REGION Network 19: DN TRR
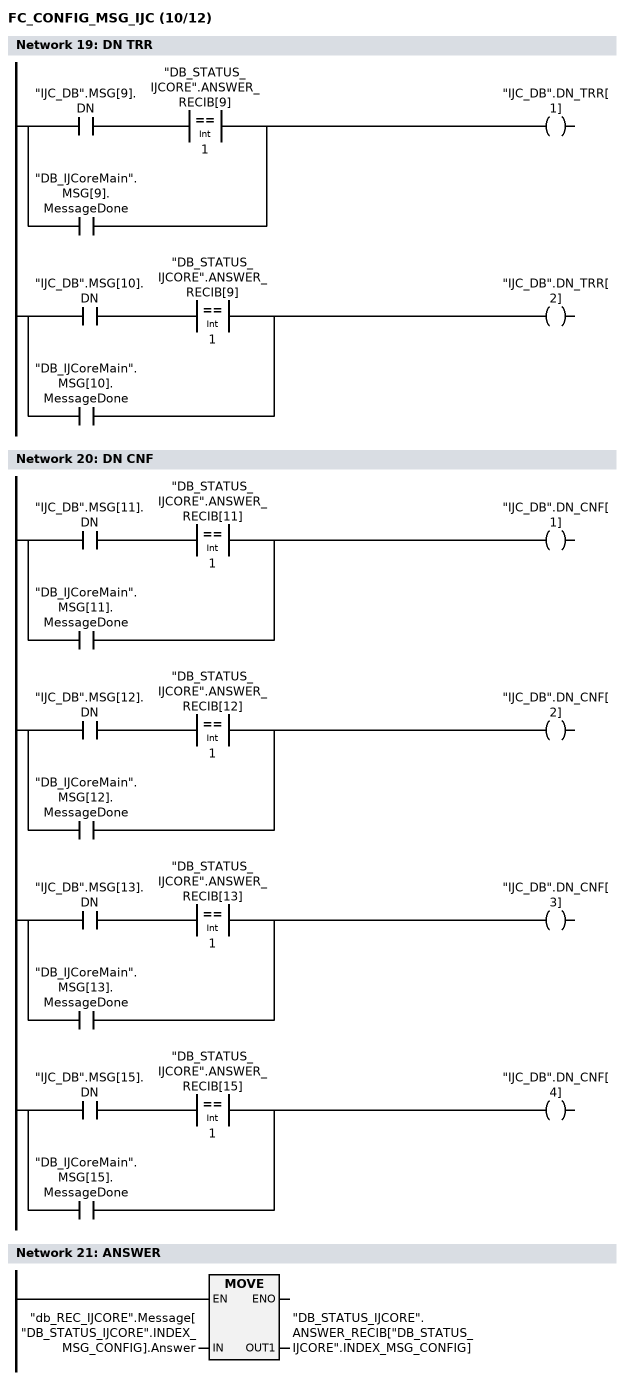
   RUNG wire#powerrail
      Contact( "IJC_DB".MSG[9].DN )
      { S7_Templates := "SrcType := Int" } EQ_Contact(in1 := "DB_STATUS_IJCORE".ANSWER_RECIB[9], in2 := 1)
      wire#w1
      Coil( "IJC_DB".DN_TRR[1] )
   END_RUNG
   RUNG wire#powerrail
      Contact( "DB_IJCoreMain".MSG[9].MessageDone )
   END_RUNG wire#w1
   RUNG wire#powerrail
      Contact( "IJC_DB".MSG[10].DN )
      { S7_Templates := "SrcType := Int" } EQ_Contact(in1 := "DB_STATUS_IJCORE".ANSWER_RECIB[9], in2 := 1)
      wire#w2
      Coil( "IJC_DB".DN_TRR[2] )
   END_RUNG
   RUNG wire#powerrail
      Contact( "DB_IJCoreMain".MSG[10].MessageDone )
   END_RUNG wire#w2
   // the same network as SCL:
   "IJC_DB".DN_TRR[1] := ("IJC_DB".MSG[9].DN AND ("DB_STATUS_IJCORE".ANSWER_RECIB[9] = 1)) OR "DB_IJCoreMain".MSG[9].MessageDone;
   "IJC_DB".DN_TRR[2] := ("IJC_DB".MSG[10].DN AND ("DB_STATUS_IJCORE".ANSWER_RECIB[9] = 1)) OR "DB_IJCoreMain".MSG[10].MessageDone;
END_REGION

REGION Network 20: DN CNF
   RUNG wire#powerrail
      Contact( "IJC_DB".MSG[11].DN )
      { S7_Templates := "SrcType := Int" } EQ_Contact(in1 := "DB_STATUS_IJCORE".ANSWER_RECIB[11], in2 := 1)
      wire#w1
      Coil( "IJC_DB".DN_CNF[1] )
   END_RUNG
   RUNG wire#powerrail
      Contact( "DB_IJCoreMain".MSG[11].MessageDone )
   END_RUNG wire#w1
   RUNG wire#powerrail
      Contact( "IJC_DB".MSG[12].DN )
      { S7_Templates := "SrcType := Int" } EQ_Contact(in1 := "DB_STATUS_IJCORE".ANSWER_RECIB[12], in2 := 1)
      wire#w2
      Coil( "IJC_DB".DN_CNF[2] )
   END_RUNG
   RUNG wire#powerrail
      Contact( "DB_IJCoreMain".MSG[12].MessageDone )
   END_RUNG wire#w2
   RUNG wire#powerrail
      Contact( "IJC_DB".MSG[13].DN )
      { S7_Templates := "SrcType := Int" } EQ_Contact(in1 := "DB_STATUS_IJCORE".ANSWER_RECIB[13], in2 := 1)
      wire#w3
      Coil( "IJC_DB".DN_CNF[3] )
   END_RUNG
   RUNG wire#powerrail
      Contact( "DB_IJCoreMain".MSG[13].MessageDone )
   END_RUNG wire#w3
   RUNG wire#powerrail
      Contact( "IJC_DB".MSG[15].DN )
      { S7_Templates := "SrcType := Int" } EQ_Contact(in1 := "DB_STATUS_IJCORE".ANSWER_RECIB[15], in2 := 1)
      wire#w4
      Coil( "IJC_DB".DN_CNF[4] )
   END_RUNG
   RUNG wire#powerrail
      Contact( "DB_IJCoreMain".MSG[15].MessageDone )
   END_RUNG wire#w4
   // the same network as SCL:
   "IJC_DB".DN_CNF[1] := ("IJC_DB".MSG[11].DN AND ("DB_STATUS_IJCORE".ANSWER_RECIB[11] = 1)) OR "DB_IJCoreMain".MSG[11].MessageDone;
   "IJC_DB".DN_CNF[2] := ("IJC_DB".MSG[12].DN AND ("DB_STATUS_IJCORE".ANSWER_RECIB[12] = 1)) OR "DB_IJCoreMain".MSG[12].MessageDone;
   "IJC_DB".DN_CNF[3] := ("IJC_DB".MSG[13].DN AND ("DB_STATUS_IJCORE".ANSWER_RECIB[13] = 1)) OR "DB_IJCoreMain".MSG[13].MessageDone;
   "IJC_DB".DN_CNF[4] := ("IJC_DB".MSG[15].DN AND ("DB_STATUS_IJCORE".ANSWER_RECIB[15] = 1)) OR "DB_IJCoreMain".MSG[15].MessageDone;
END_REGION

REGION Network 21: ANSWER
   RUNG wire#powerrail
      Move(in := "db_REC_IJCORE".Message["DB_STATUS_IJCORE".INDEX_MSG_CONFIG].Answer, out1 => "DB_STATUS_IJCORE".ANSWER_RECIB["DB_STATUS_IJCORE".INDEX_MSG_CONFIG])
   END_RUNG
   // the same network as SCL:
   "DB_STATUS_IJCORE".ANSWER_RECIB["DB_STATUS_IJCORE".INDEX_MSG_CONFIG] := "db_REC_IJCORE".Message["DB_STATUS_IJCORE".INDEX_MSG_CONFIG].Answer;
END_REGION

REGION Network 22: ANSWER NFP
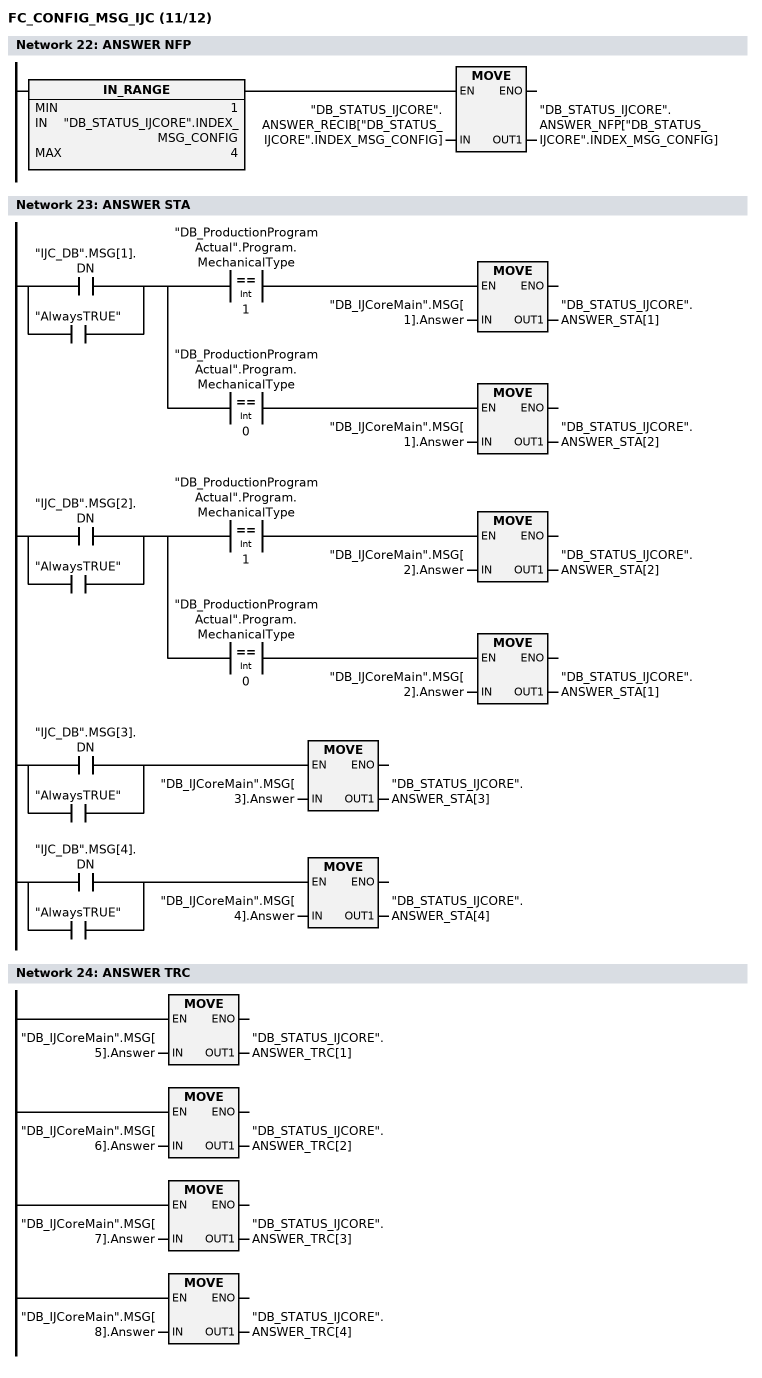
   RUNG wire#powerrail
      { S7_Templates := "SrcType := DInt" } InRange(min := 1, in := "DB_STATUS_IJCORE".INDEX_MSG_CONFIG, max := 4)
      Move(in := "DB_STATUS_IJCORE".ANSWER_RECIB["DB_STATUS_IJCORE".INDEX_MSG_CONFIG], out1 => "DB_STATUS_IJCORE".ANSWER_NFP["DB_STATUS_IJCORE".INDEX_MSG_CONFIG])
   END_RUNG
   // the same network as SCL:
   IF (1 <= "DB_STATUS_IJCORE".INDEX_MSG_CONFIG) AND ("DB_STATUS_IJCORE".INDEX_MSG_CONFIG <= 4) THEN
       "DB_STATUS_IJCORE".ANSWER_NFP["DB_STATUS_IJCORE".INDEX_MSG_CONFIG] := "DB_STATUS_IJCORE".ANSWER_RECIB["DB_STATUS_IJCORE".INDEX_MSG_CONFIG];
   END_IF;
END_REGION

REGION Network 23: ANSWER STA
   RUNG wire#powerrail
      Contact( "IJC_DB".MSG[1].DN )
      wire#w1
      { S7_Templates := "SrcType := Int" } EQ_Contact(in1 := "DB_ProductionProgramActual".Program.MechanicalType, in2 := 1)
      Move(in := "DB_IJCoreMain".MSG[1].Answer, out1 => "DB_STATUS_IJCORE".ANSWER_STA[1])
   END_RUNG
   RUNG wire#powerrail
      Contact( "AlwaysTRUE" )
   END_RUNG wire#w1
   RUNG wire#w1
      { S7_Templates := "SrcType := Int" } EQ_Contact(in1 := "DB_ProductionProgramActual".Program.MechanicalType, in2 := 0)
      Move(in := "DB_IJCoreMain".MSG[1].Answer, out1 => "DB_STATUS_IJCORE".ANSWER_STA[2])
   END_RUNG
   RUNG wire#powerrail
      Contact( "IJC_DB".MSG[2].DN )
      wire#w2
      { S7_Templates := "SrcType := Int" } EQ_Contact(in1 := "DB_ProductionProgramActual".Program.MechanicalType, in2 := 1)
      Move(in := "DB_IJCoreMain".MSG[2].Answer, out1 => "DB_STATUS_IJCORE".ANSWER_STA[2])
   END_RUNG
   RUNG wire#powerrail
      Contact( "AlwaysTRUE" )
   END_RUNG wire#w2
   RUNG wire#w2
      { S7_Templates := "SrcType := Int" } EQ_Contact(in1 := "DB_ProductionProgramActual".Program.MechanicalType, in2 := 0)
      Move(in := "DB_IJCoreMain".MSG[2].Answer, out1 => "DB_STATUS_IJCORE".ANSWER_STA[1])
   END_RUNG
   RUNG wire#powerrail
      Contact( "IJC_DB".MSG[3].DN )
      wire#w3
      Move(in := "DB_IJCoreMain".MSG[3].Answer, out1 => "DB_STATUS_IJCORE".ANSWER_STA[3])
   END_RUNG
   RUNG wire#powerrail
      Contact( "AlwaysTRUE" )
   END_RUNG wire#w3
   RUNG wire#powerrail
      Contact( "IJC_DB".MSG[4].DN )
      wire#w4
      Move(in := "DB_IJCoreMain".MSG[4].Answer, out1 => "DB_STATUS_IJCORE".ANSWER_STA[4])
   END_RUNG
   RUNG wire#powerrail
      Contact( "AlwaysTRUE" )
   END_RUNG wire#w4
   // the same network as SCL:
   #_w1 := "IJC_DB".MSG[1].DN OR "AlwaysTRUE";
   IF #_w1 AND ("DB_ProductionProgramActual".Program.MechanicalType = 1) THEN
       "DB_STATUS_IJCORE".ANSWER_STA[1] := "DB_IJCoreMain".MSG[1].Answer;
   END_IF;
   IF #_w1 AND ("DB_ProductionProgramActual".Program.MechanicalType = 0) THEN
       "DB_STATUS_IJCORE".ANSWER_STA[2] := "DB_IJCoreMain".MSG[1].Answer;
   END_IF;
   #_w2 := "IJC_DB".MSG[2].DN OR "AlwaysTRUE";
   IF #_w2 AND ("DB_ProductionProgramActual".Program.MechanicalType = 1) THEN
       "DB_STATUS_IJCORE".ANSWER_STA[2] := "DB_IJCoreMain".MSG[2].Answer;
   END_IF;
   IF #_w2 AND ("DB_ProductionProgramActual".Program.MechanicalType = 0) THEN
       "DB_STATUS_IJCORE".ANSWER_STA[1] := "DB_IJCoreMain".MSG[2].Answer;
   END_IF;
   IF "IJC_DB".MSG[3].DN OR "AlwaysTRUE" THEN
       "DB_STATUS_IJCORE".ANSWER_STA[3] := "DB_IJCoreMain".MSG[3].Answer;
   END_IF;
   IF "IJC_DB".MSG[4].DN OR "AlwaysTRUE" THEN
       "DB_STATUS_IJCORE".ANSWER_STA[4] := "DB_IJCoreMain".MSG[4].Answer;
   END_IF;
END_REGION

REGION Network 24: ANSWER TRC
   RUNG wire#powerrail
      Move(in := "DB_IJCoreMain".MSG[5].Answer, out1 => "DB_STATUS_IJCORE".ANSWER_TRC[1])
   END_RUNG
   RUNG wire#powerrail
      Move(in := "DB_IJCoreMain".MSG[6].Answer, out1 => "DB_STATUS_IJCORE".ANSWER_TRC[2])
   END_RUNG
   RUNG wire#powerrail
      Move(in := "DB_IJCoreMain".MSG[7].Answer, out1 => "DB_STATUS_IJCORE".ANSWER_TRC[3])
   END_RUNG
   RUNG wire#powerrail
      Move(in := "DB_IJCoreMain".MSG[8].Answer, out1 => "DB_STATUS_IJCORE".ANSWER_TRC[4])
   END_RUNG
   // the same network as SCL:
   "DB_STATUS_IJCORE".ANSWER_TRC[1] := "DB_IJCoreMain".MSG[5].Answer;
   "DB_STATUS_IJCORE".ANSWER_TRC[2] := "DB_IJCoreMain".MSG[6].Answer;
   "DB_STATUS_IJCORE".ANSWER_TRC[3] := "DB_IJCoreMain".MSG[7].Answer;
   "DB_STATUS_IJCORE".ANSWER_TRC[4] := "DB_IJCoreMain".MSG[8].Answer;
END_REGION

REGION Network 25: STATUS MSG TRC
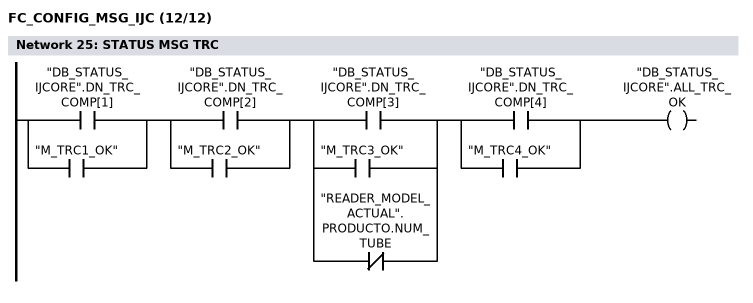
   RUNG wire#powerrail
      Contact( "DB_STATUS_IJCORE".DN_TRC_COMP[1] )
      wire#w1
      Contact( "DB_STATUS_IJCORE".DN_TRC_COMP[2] )
      wire#w2
      Contact( "DB_STATUS_IJCORE".DN_TRC_COMP[3] )
      wire#w3
      Contact( "DB_STATUS_IJCORE".DN_TRC_COMP[4] )
      wire#w4
      Coil( "DB_STATUS_IJCORE".ALL_TRC_OK )
   END_RUNG
   RUNG wire#powerrail
      Contact( "M_TRC1_OK" )
   END_RUNG wire#w1
   RUNG wire#w1
      Contact( "M_TRC2_OK" )
   END_RUNG wire#w2
   RUNG wire#w2
      Contact( "M_TRC3_OK" )
   END_RUNG wire#w3
   RUNG wire#w2
      I_Contact( "READER_MODEL_ACTUAL".PRODUCTO.NUM_TUBE )
   END_RUNG wire#w3
   RUNG wire#w3
      Contact( "M_TRC4_OK" )
   END_RUNG wire#w4
   // the same network as SCL:
   "DB_STATUS_IJCORE".ALL_TRC_OK := ("DB_STATUS_IJCORE".DN_TRC_COMP[1] OR "M_TRC1_OK") AND ("DB_STATUS_IJCORE".DN_TRC_COMP[2] OR "M_TRC2_OK") AND ("DB_STATUS_IJCORE".DN_TRC_COMP[3] OR "M_TRC3_OK" OR NOT "READER_MODEL_ACTUAL".PRODUCTO.NUM_TUBE) AND ("DB_STATUS_IJCORE".DN_TRC_COMP[4] OR "M_TRC4_OK");
END_REGION
END_FUNCTION

FUNCTION_BLOCK "AWAKE_SIGNAL"   // FB1002, LAD
TITLE = Awake signal
{ S7_Optimized_Access := 'TRUE' }
VERSION : 0.1
// This function supervise Awake signal, 
// - Awake signal is to test communication between PLC and IJCORE. 
// - Awake signal is set to 1 by PLC and set to -1 by IJCORE alternatively.
// - first PLC check if awake signal is different of 1, if it is, PLC launch timer T1 
//  (1s<T1<10s). at the end of this temporisation, PLC set awake signal to 1 and 
//  launch Timer 2. 
// - if IJCORE don't set awake signal to -1 before the end of timer 2,PLC generate  
//   Time out fault for awake signal.
// stored: AutoNumber false, IsIECCheckEnabled false, IsRetainMemResEnabled false, MemoryReserve 100, SetENOAutomatically false, UDAEnableTagReadback false
   VAR_INPUT
      ack_error : Bool;   // Acknowledge button
   END_VAR
   VAR_OUTPUT
      State_com : SInt;   // State of communication : 0 no communication 1: communication lost 2 : good communication
   END_VAR
   VAR RETAIN
      T1PresetValue : Time := T#1S;   // Bit of life Timer 1 preset value
      T2PresetValue : Time := T#60S;   // Bit of Life Timer 2 preset value
   END_VAR
   VAR
      AwSignalTimeOutFault : Bool := 0;   // Awake signal time out fault
      Reset_Counters : Bool;   // Signal to reset counter
      Restart_Counter_bit_of_life : USInt := 0;   // Number of restart bit of life
      NB_Bit_of_Life : Bool;   // Number bit of life
      number_restart : DInt;   // Number restart communication
      check_restart : Bool;   // Memo to check restart communication
      t13 : TON_TIME;
      t16 { S7_SetPoint := 'True'} : TON_TIME;
      t5 { S7_SetPoint := 'True'} : TON_TIME;
      t4 { S7_SetPoint := 'True'} : TON_TIME;
   END_VAR
   VAR CONSTANT
      Trestart : Time := T#200ms;   // Timer when IJCore replies normally
      T3 : Time := T#2s;   // Timer when IJCore blocks a short period of time
   END_VAR
   VAR_TEMP   // added for the SCL form of the ladder/FBD networks
      _w1 : Bool;
   END_VAR
BEGIN

REGION Network 1: - if awake signal is -1 then launch timer 1
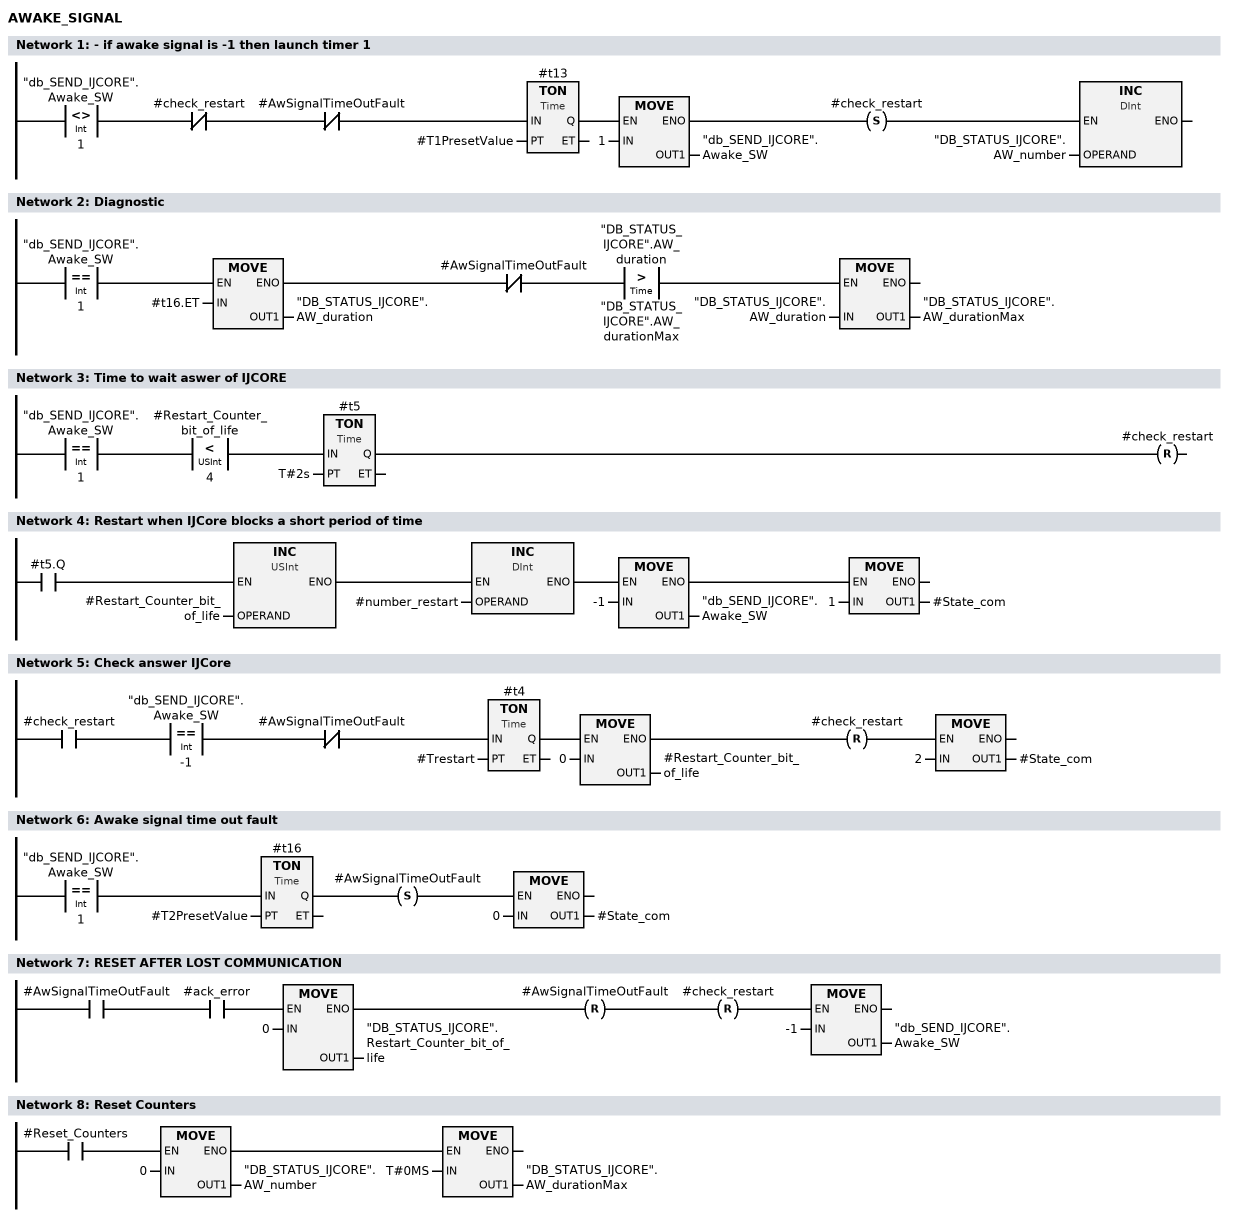
   RUNG wire#powerrail
      { S7_Templates := "SrcType := Int" } NE_Contact(in1 := "db_SEND_IJCORE".Awake_SW, in2 := 1)
      I_Contact( #check_restart )
      I_Contact( #AwSignalTimeOutFault )
      { S7_Templates := "time_type := Time" } #t13.TON(pt := #T1PresetValue, et =>)
      Move(in := 1, out1 => "db_SEND_IJCORE".Awake_SW)
      S_Coil( #check_restart )
      { S7_Templates := "DestType := DInt" } Inc( "DB_STATUS_IJCORE".AW_number )
   END_RUNG
   // the same network as SCL:
   #t13(IN := ("db_SEND_IJCORE".Awake_SW <> 1) AND NOT #check_restart AND NOT #AwSignalTimeOutFault,   // TON
        PT := #T1PresetValue);
   IF #t13.Q THEN
       "db_SEND_IJCORE".Awake_SW := 1;
       #check_restart := TRUE;
       "DB_STATUS_IJCORE".AW_number := "DB_STATUS_IJCORE".AW_number + 1;
   END_IF;
END_REGION

REGION Network 2: Diagnostic
   RUNG wire#powerrail
      { S7_Templates := "SrcType := Int" } EQ_Contact(in1 := "db_SEND_IJCORE".Awake_SW, in2 := 1)
      Move(in := #t16.ET, out1 => "DB_STATUS_IJCORE".AW_duration)
      I_Contact( #AwSignalTimeOutFault )
      { S7_Templates := "SrcType := Time" } GT_Contact(in1 := "DB_STATUS_IJCORE".AW_duration, in2 := "DB_STATUS_IJCORE".AW_durationMax)
      Move(in := "DB_STATUS_IJCORE".AW_duration, out1 => "DB_STATUS_IJCORE".AW_durationMax)
   END_RUNG
   // the same network as SCL:
   #_w1 := "db_SEND_IJCORE".Awake_SW = 1;
   IF #_w1 THEN "DB_STATUS_IJCORE".AW_duration := #t16.ET; END_IF;
   IF #_w1 AND NOT #AwSignalTimeOutFault AND ("DB_STATUS_IJCORE".AW_duration > "DB_STATUS_IJCORE".AW_durationMax) THEN
       "DB_STATUS_IJCORE".AW_durationMax := "DB_STATUS_IJCORE".AW_duration;
   END_IF;
END_REGION

REGION Network 3: Time to wait aswer of IJCORE
   RUNG wire#powerrail
      { S7_Templates := "SrcType := Int" } EQ_Contact(in1 := "db_SEND_IJCORE".Awake_SW, in2 := 1)
      { S7_Templates := "SrcType := USInt" } LT_Contact(in1 := #Restart_Counter_bit_of_life, in2 := 4)
      { S7_Templates := "time_type := Time" } #t5.TON(pt := T#2s, et =>)
      R_Coil( #check_restart )
   END_RUNG
   // the same network as SCL:
   #t5(IN := ("db_SEND_IJCORE".Awake_SW = 1) AND (#Restart_Counter_bit_of_life < 4), PT := T#2s);   // TON
   IF #t5.Q THEN #check_restart := FALSE; END_IF;
END_REGION

REGION Network 4: Restart when IJCore blocks a short period of time
   RUNG wire#powerrail
      Contact( #t5.Q )
      { S7_Templates := "DestType := USInt" } Inc( #Restart_Counter_bit_of_life )
      { S7_Templates := "DestType := DInt" } Inc( #number_restart )
      Move(in := -1, out1 => "db_SEND_IJCORE".Awake_SW)
      Move(in := 1, out1 => #State_com)
   END_RUNG
   // the same network as SCL:
   IF #t5.Q THEN
       #Restart_Counter_bit_of_life := #Restart_Counter_bit_of_life + 1;
       #number_restart := #number_restart + 1;
       "db_SEND_IJCORE".Awake_SW := -1;
       #State_com := 1;
   END_IF;
END_REGION

REGION Network 5: Check answer IJCore
   RUNG wire#powerrail
      Contact( #check_restart )
      { S7_Templates := "SrcType := Int" } EQ_Contact(in1 := "db_SEND_IJCORE".Awake_SW, in2 := -1)
      I_Contact( #AwSignalTimeOutFault )
      { S7_Templates := "time_type := Time" } #t4.TON(pt := #Trestart, et =>)
      Move(in := 0, out1 => #Restart_Counter_bit_of_life)
      R_Coil( #check_restart )
      Move(in := 2, out1 => #State_com)
   END_RUNG
   // the same network as SCL:
   #t4(IN := #check_restart AND ("db_SEND_IJCORE".Awake_SW = (-1)) AND NOT #AwSignalTimeOutFault,   // TON
       PT := #Trestart);
   IF #t4.Q THEN
       #Restart_Counter_bit_of_life := 0;
       #check_restart := FALSE;
       #State_com := 2;
   END_IF;
END_REGION

REGION Network 6: Awake signal time out fault
   RUNG wire#powerrail
      { S7_Templates := "SrcType := Int" } EQ_Contact(in1 := "db_SEND_IJCORE".Awake_SW, in2 := 1)
      { S7_Templates := "time_type := Time" } #t16.TON(pt := #T2PresetValue, et =>)
      S_Coil( #AwSignalTimeOutFault )
      Move(in := 0, out1 => #State_com)
   END_RUNG
   // the same network as SCL:
   #t16(IN := "db_SEND_IJCORE".Awake_SW = 1, PT := #T2PresetValue);   // TON
   IF #t16.Q THEN
       #AwSignalTimeOutFault := TRUE;
       #State_com := 0;
   END_IF;
END_REGION

REGION Network 7: RESET AFTER LOST COMMUNICATION
   RUNG wire#powerrail
      Contact( #AwSignalTimeOutFault )
      Contact( #ack_error )
      Move(in := 0, out1 => "DB_STATUS_IJCORE".Restart_Counter_bit_of_life)
      R_Coil( #AwSignalTimeOutFault )
      R_Coil( #check_restart )
      Move(in := -1, out1 => "db_SEND_IJCORE".Awake_SW)
   END_RUNG
   // the same network as SCL:
   IF #AwSignalTimeOutFault AND #ack_error THEN "DB_STATUS_IJCORE".Restart_Counter_bit_of_life := 0; END_IF;
   #_w1 := #AwSignalTimeOutFault AND #ack_error;
   IF #_w1 THEN
       #AwSignalTimeOutFault := FALSE;
       #check_restart := FALSE;
       "db_SEND_IJCORE".Awake_SW := -1;
   END_IF;
END_REGION

REGION Network 8: Reset Counters
   RUNG wire#powerrail
      Contact( #Reset_Counters )
      Move(in := 0, out1 => "DB_STATUS_IJCORE".AW_number)
      Move(in := T#0MS, out1 => "DB_STATUS_IJCORE".AW_durationMax)
   END_RUNG
   // the same network as SCL:
   IF #Reset_Counters THEN
       "DB_STATUS_IJCORE".AW_number := 0;
       "DB_STATUS_IJCORE".AW_durationMax := T#0MS;
   END_IF;
END_REGION
END_FUNCTION_BLOCK

FUNCTION_BLOCK "IJCoreMain"   // FB1000, LAD
TITLE = IJCore Main
{ S7_Optimized_Access := 'TRUE' }
VERSION : 0.1
// stored: AutoNumber false, IsIECCheckEnabled false, IsRetainMemResEnabled false, MemoryReserve 100, SetENOAutomatically false, UDAEnableTagReadback false
   VAR
      Enable : Bool;
      Mode : UInt;
      Indicator : Int;
      AlarmReset : Bool;
      AWAKE_SIGNAL { S7_SetPoint := 'True'} : "AWAKE_SIGNAL";
      MSG : Array[1..20] of "IJCoreMessageProcotol";
      NFP { S7_SetPoint := 'True'} : Array[1..4] of String[30];
   END_VAR
   VAR_TEMP
      MessageDone : Bool;
      Answer : DInt;
      Fault : DInt;
   END_VAR
   VAR CONSTANT
      STA : Int := 5;
      CNF : Int := 1;
      TRC : Int := 13;
      PFC : Int := 9;
      TRR : Int := 7;
   END_VAR
BEGIN

REGION Network 1
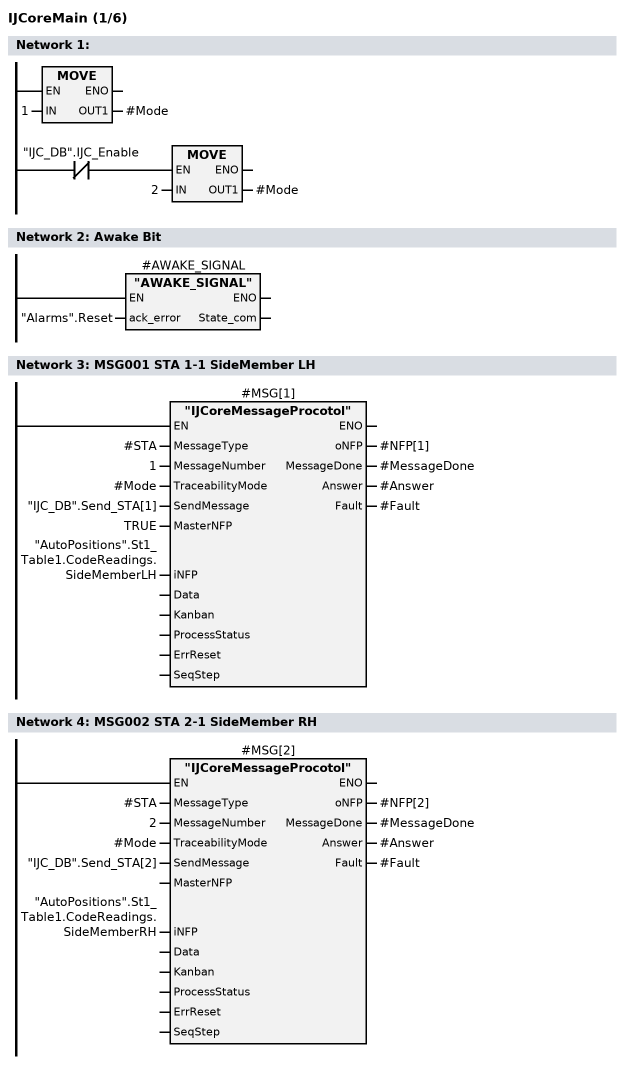
   RUNG wire#powerrail
      Move(in := 1, out1 => #Mode)
   END_RUNG
   RUNG wire#powerrail
      I_Contact( "IJC_DB".IJC_Enable )
      Move(in := 2, out1 => #Mode)
   END_RUNG
   // the same network as SCL:
   #Mode := 1;
   IF NOT "IJC_DB".IJC_Enable THEN #Mode := 2; END_IF;
END_REGION

REGION Network 2: Awake Bit
   RUNG wire#powerrail
      #AWAKE_SIGNAL(ack_error := "Alarms".Reset, State_com =>)
   END_RUNG
   // the same network as SCL:
   #AWAKE_SIGNAL(ack_error := "Alarms".Reset);   // "AWAKE_SIGNAL"
END_REGION

REGION Network 3: MSG001 STA 1-1 SideMember LH
   RUNG wire#powerrail
      #MSG[1](MessageType := #STA, MessageNumber := 1, TraceabilityMode := #Mode, SendMessage := "IJC_DB".Send_STA[1], MasterNFP := TRUE, iNFP := "AutoPositions".St1_Table1.CodeReadings.SideMemberLH, Data :=, Kanban :=, ProcessStatus :=, ErrReset :=, SeqStep :=, oNFP => #NFP[1], MessageDone => #MessageDone, Answer => #Answer, Fault => #Fault)
   END_RUNG
   // the same network as SCL:
   #MSG[1](MessageType := #STA,   // "IJCoreMessageProcotol"
           MessageNumber := 1,
           TraceabilityMode := #Mode,
           SendMessage := "IJC_DB".Send_STA[1],
           MasterNFP := TRUE,
           iNFP := "AutoPositions".St1_Table1.CodeReadings.SideMemberLH,
           oNFP => #NFP[1],
           MessageDone => #MessageDone,
           Answer => #Answer,
           Fault => #Fault);
END_REGION

REGION Network 4: MSG002 STA 2-1 SideMember RH
   RUNG wire#powerrail
      #MSG[2](MessageType := #STA, MessageNumber := 2, TraceabilityMode := #Mode, SendMessage := "IJC_DB".Send_STA[2], MasterNFP :=, iNFP := "AutoPositions".St1_Table1.CodeReadings.SideMemberRH, Data :=, Kanban :=, ProcessStatus :=, ErrReset :=, SeqStep :=, oNFP => #NFP[2], MessageDone => #MessageDone, Answer => #Answer, Fault => #Fault)
   END_RUNG
   // the same network as SCL:
   #MSG[2](MessageType := #STA,   // "IJCoreMessageProcotol"
           MessageNumber := 2,
           TraceabilityMode := #Mode,
           SendMessage := "IJC_DB".Send_STA[2],
           iNFP := "AutoPositions".St1_Table1.CodeReadings.SideMemberRH,
           oNFP => #NFP[2],
           MessageDone => #MessageDone,
           Answer => #Answer,
           Fault => #Fault);
END_REGION

REGION Network 5: MSG003 STA 3-1 Front Tube
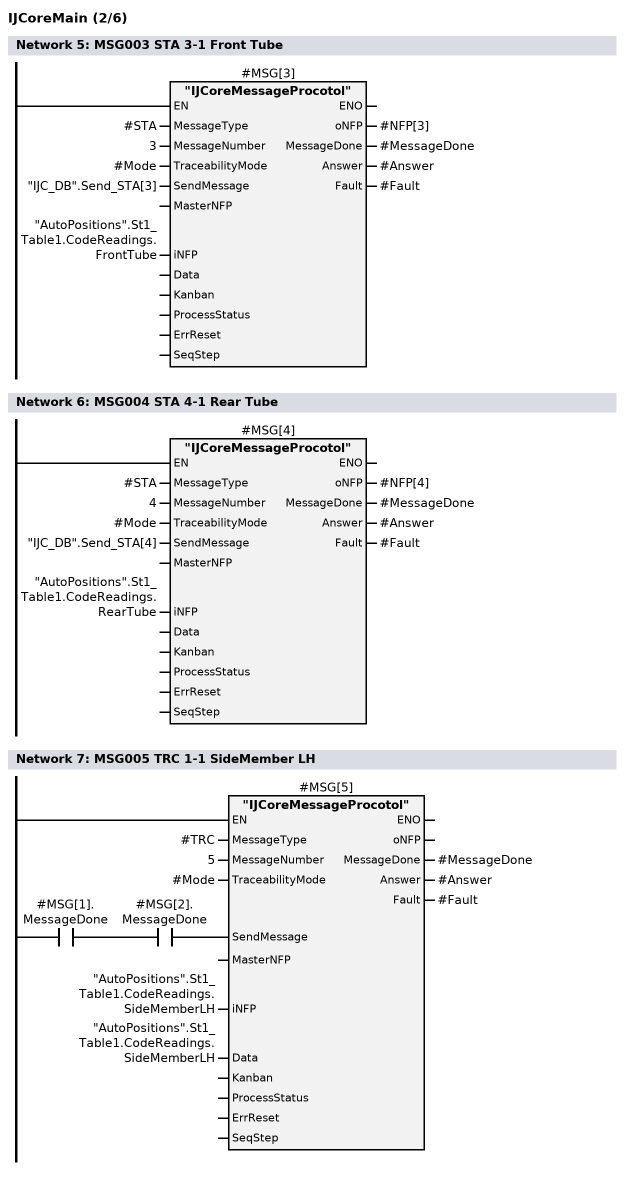
   RUNG wire#powerrail
      #MSG[3](MessageType := #STA, MessageNumber := 3, TraceabilityMode := #Mode, SendMessage := "IJC_DB".Send_STA[3], MasterNFP :=, iNFP := "AutoPositions".St1_Table1.CodeReadings.FrontTube, Data :=, Kanban :=, ProcessStatus :=, ErrReset :=, SeqStep :=, oNFP => #NFP[3], MessageDone => #MessageDone, Answer => #Answer, Fault => #Fault)
   END_RUNG
   // the same network as SCL:
   #MSG[3](MessageType := #STA,   // "IJCoreMessageProcotol"
           MessageNumber := 3,
           TraceabilityMode := #Mode,
           SendMessage := "IJC_DB".Send_STA[3],
           iNFP := "AutoPositions".St1_Table1.CodeReadings.FrontTube,
           oNFP => #NFP[3],
           MessageDone => #MessageDone,
           Answer => #Answer,
           Fault => #Fault);
END_REGION

REGION Network 6: MSG004 STA 4-1 Rear Tube
   RUNG wire#powerrail
      #MSG[4](MessageType := #STA, MessageNumber := 4, TraceabilityMode := #Mode, SendMessage := "IJC_DB".Send_STA[4], MasterNFP :=, iNFP := "AutoPositions".St1_Table1.CodeReadings.RearTube, Data :=, Kanban :=, ProcessStatus :=, ErrReset :=, SeqStep :=, oNFP => #NFP[4], MessageDone => #MessageDone, Answer => #Answer, Fault => #Fault)
   END_RUNG
   // the same network as SCL:
   #MSG[4](MessageType := #STA,   // "IJCoreMessageProcotol"
           MessageNumber := 4,
           TraceabilityMode := #Mode,
           SendMessage := "IJC_DB".Send_STA[4],
           iNFP := "AutoPositions".St1_Table1.CodeReadings.RearTube,
           oNFP => #NFP[4],
           MessageDone => #MessageDone,
           Answer => #Answer,
           Fault => #Fault);
END_REGION

REGION Network 7: MSG005 TRC 1-1 SideMember LH
   RUNG wire#powerrail
      #MSG[5](SendMessage := wire#w1, MessageType := #TRC, MessageNumber := 5, TraceabilityMode := #Mode, MasterNFP :=, iNFP := "AutoPositions".St1_Table1.CodeReadings.SideMemberLH, Data := "AutoPositions".St1_Table1.CodeReadings.SideMemberLH, Kanban :=, ProcessStatus :=, ErrReset :=, SeqStep :=, oNFP =>, MessageDone => #MessageDone, Answer => #Answer, Fault => #Fault)
   END_RUNG
   RUNG wire#powerrail
      Contact( #MSG[1].MessageDone )
      Contact( #MSG[2].MessageDone )
   END_RUNG wire#w1
   // the same network as SCL:
   #MSG[5](MessageType := #TRC,   // "IJCoreMessageProcotol"
           MessageNumber := 5,
           TraceabilityMode := #Mode,
           SendMessage := #MSG[1].MessageDone AND #MSG[2].MessageDone,
           iNFP := "AutoPositions".St1_Table1.CodeReadings.SideMemberLH,
           Data := "AutoPositions".St1_Table1.CodeReadings.SideMemberLH,
           MessageDone => #MessageDone,
           Answer => #Answer,
           Fault => #Fault);
END_REGION

REGION Network 8: MSG006 TRC 1-2 SideMember RH
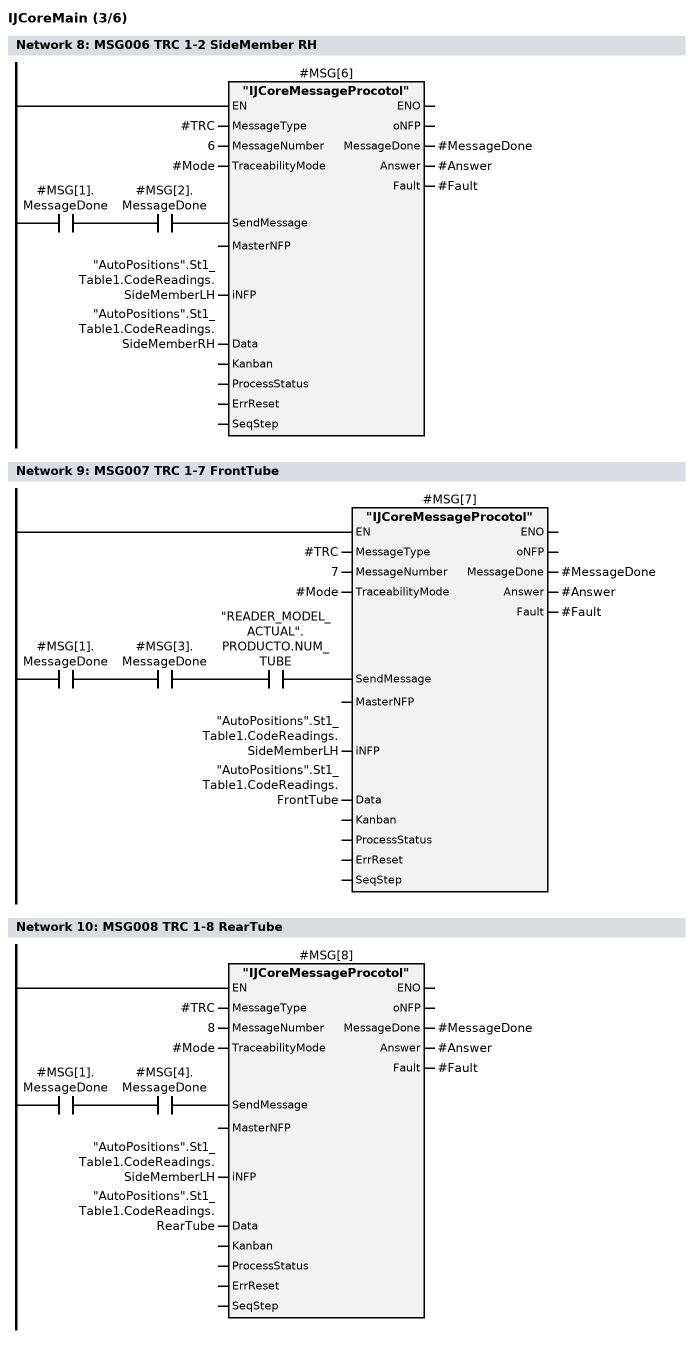
   RUNG wire#powerrail
      #MSG[6](SendMessage := wire#w1, MessageType := #TRC, MessageNumber := 6, TraceabilityMode := #Mode, MasterNFP :=, iNFP := "AutoPositions".St1_Table1.CodeReadings.SideMemberLH, Data := "AutoPositions".St1_Table1.CodeReadings.SideMemberRH, Kanban :=, ProcessStatus :=, ErrReset :=, SeqStep :=, oNFP =>, MessageDone => #MessageDone, Answer => #Answer, Fault => #Fault)
   END_RUNG
   RUNG wire#powerrail
      Contact( #MSG[1].MessageDone )
      Contact( #MSG[2].MessageDone )
   END_RUNG wire#w1
   // the same network as SCL:
   #MSG[6](MessageType := #TRC,   // "IJCoreMessageProcotol"
           MessageNumber := 6,
           TraceabilityMode := #Mode,
           SendMessage := #MSG[1].MessageDone AND #MSG[2].MessageDone,
           iNFP := "AutoPositions".St1_Table1.CodeReadings.SideMemberLH,
           Data := "AutoPositions".St1_Table1.CodeReadings.SideMemberRH,
           MessageDone => #MessageDone,
           Answer => #Answer,
           Fault => #Fault);
END_REGION

REGION Network 9: MSG007 TRC 1-7 FrontTube
   RUNG wire#powerrail
      #MSG[7](SendMessage := wire#w1, MessageType := #TRC, MessageNumber := 7, TraceabilityMode := #Mode, MasterNFP :=, iNFP := "AutoPositions".St1_Table1.CodeReadings.SideMemberLH, Data := "AutoPositions".St1_Table1.CodeReadings.FrontTube, Kanban :=, ProcessStatus :=, ErrReset :=, SeqStep :=, oNFP =>, MessageDone => #MessageDone, Answer => #Answer, Fault => #Fault)
   END_RUNG
   RUNG wire#powerrail
      Contact( #MSG[1].MessageDone )
      Contact( #MSG[3].MessageDone )
      Contact( "READER_MODEL_ACTUAL".PRODUCTO.NUM_TUBE )
   END_RUNG wire#w1
   // the same network as SCL:
   #MSG[7](MessageType := #TRC,   // "IJCoreMessageProcotol"
           MessageNumber := 7,
           TraceabilityMode := #Mode,
           SendMessage := #MSG[1].MessageDone AND #MSG[3].MessageDone AND "READER_MODEL_ACTUAL".PRODUCTO.NUM_TUBE,
           iNFP := "AutoPositions".St1_Table1.CodeReadings.SideMemberLH,
           Data := "AutoPositions".St1_Table1.CodeReadings.FrontTube,
           MessageDone => #MessageDone,
           Answer => #Answer,
           Fault => #Fault);
END_REGION

REGION Network 10: MSG008 TRC 1-8 RearTube
   RUNG wire#powerrail
      #MSG[8](SendMessage := wire#w1, MessageType := #TRC, MessageNumber := 8, TraceabilityMode := #Mode, MasterNFP :=, iNFP := "AutoPositions".St1_Table1.CodeReadings.SideMemberLH, Data := "AutoPositions".St1_Table1.CodeReadings.RearTube, Kanban :=, ProcessStatus :=, ErrReset :=, SeqStep :=, oNFP =>, MessageDone => #MessageDone, Answer => #Answer, Fault => #Fault)
   END_RUNG
   RUNG wire#powerrail
      Contact( #MSG[1].MessageDone )
      Contact( #MSG[4].MessageDone )
   END_RUNG wire#w1
   // the same network as SCL:
   #MSG[8](MessageType := #TRC,   // "IJCoreMessageProcotol"
           MessageNumber := 8,
           TraceabilityMode := #Mode,
           SendMessage := #MSG[1].MessageDone AND #MSG[4].MessageDone,
           iNFP := "AutoPositions".St1_Table1.CodeReadings.SideMemberLH,
           Data := "AutoPositions".St1_Table1.CodeReadings.RearTube,
           MessageDone => #MessageDone,
           Answer => #Answer,
           Fault => #Fault);
END_REGION

REGION Network 11: MSG009 TRR 1-1 Results of riveting
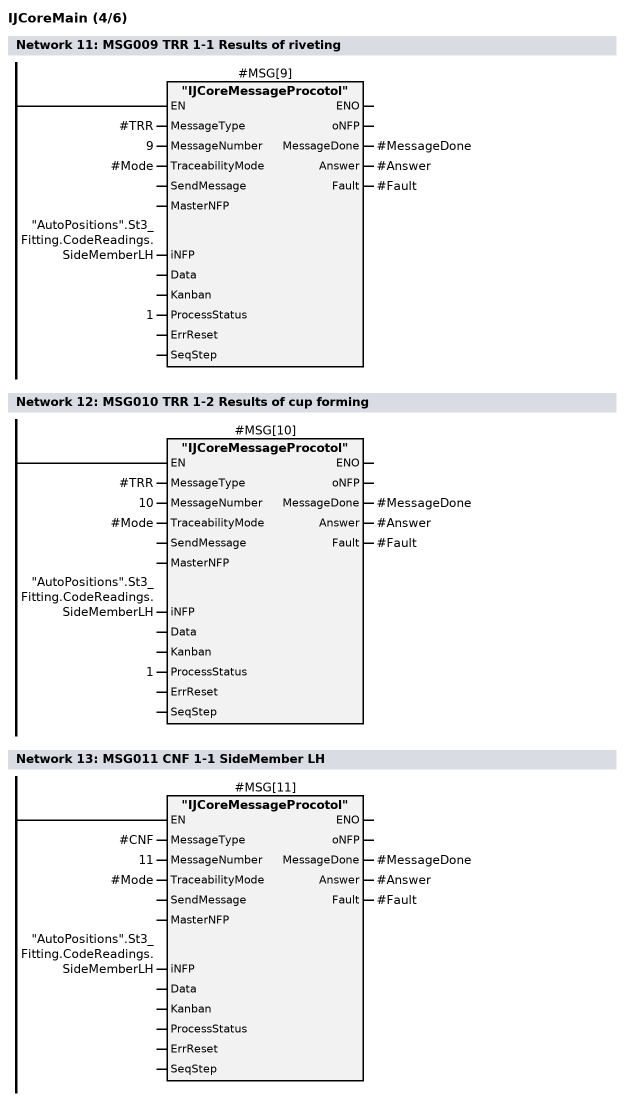
   RUNG wire#powerrail
      #MSG[9](MessageType := #TRR, MessageNumber := 9, TraceabilityMode := #Mode, SendMessage :=, MasterNFP :=, iNFP := "AutoPositions".St3_Fitting.CodeReadings.SideMemberLH, Data :=, Kanban :=, ProcessStatus := 1, ErrReset :=, SeqStep :=, oNFP =>, MessageDone => #MessageDone, Answer => #Answer, Fault => #Fault)
   END_RUNG
   // the same network as SCL:
   #MSG[9](MessageType := #TRR,   // "IJCoreMessageProcotol"
           MessageNumber := 9,
           TraceabilityMode := #Mode,
           iNFP := "AutoPositions".St3_Fitting.CodeReadings.SideMemberLH,
           ProcessStatus := 1,
           MessageDone => #MessageDone,
           Answer => #Answer,
           Fault => #Fault);
END_REGION

REGION Network 12: MSG010 TRR 1-2 Results of cup forming
   RUNG wire#powerrail
      #MSG[10](MessageType := #TRR, MessageNumber := 10, TraceabilityMode := #Mode, SendMessage :=, MasterNFP :=, iNFP := "AutoPositions".St3_Fitting.CodeReadings.SideMemberLH, Data :=, Kanban :=, ProcessStatus := 1, ErrReset :=, SeqStep :=, oNFP =>, MessageDone => #MessageDone, Answer => #Answer, Fault => #Fault)
   END_RUNG
   // the same network as SCL:
   #MSG[10](MessageType := #TRR,   // "IJCoreMessageProcotol"
            MessageNumber := 10,
            TraceabilityMode := #Mode,
            iNFP := "AutoPositions".St3_Fitting.CodeReadings.SideMemberLH,
            ProcessStatus := 1,
            MessageDone => #MessageDone,
            Answer => #Answer,
            Fault => #Fault);
END_REGION

REGION Network 13: MSG011 CNF 1-1 SideMember LH
   RUNG wire#powerrail
      #MSG[11](MessageType := #CNF, MessageNumber := 11, TraceabilityMode := #Mode, SendMessage :=, MasterNFP :=, iNFP := "AutoPositions".St3_Fitting.CodeReadings.SideMemberLH, Data :=, Kanban :=, ProcessStatus :=, ErrReset :=, SeqStep :=, oNFP =>, MessageDone => #MessageDone, Answer => #Answer, Fault => #Fault)
   END_RUNG
   // the same network as SCL:
   #MSG[11](MessageType := #CNF,   // "IJCoreMessageProcotol"
            MessageNumber := 11,
            TraceabilityMode := #Mode,
            iNFP := "AutoPositions".St3_Fitting.CodeReadings.SideMemberLH,
            MessageDone => #MessageDone,
            Answer => #Answer,
            Fault => #Fault);
END_REGION

REGION Network 14: MSG012 CNF 1-2 SideMember RH
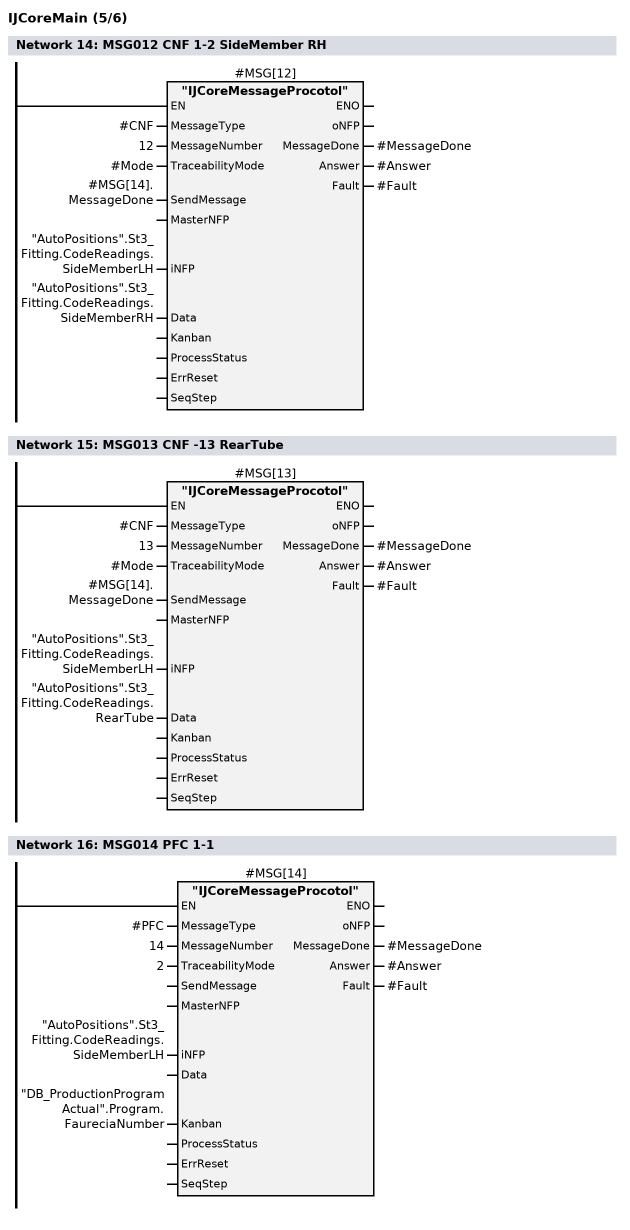
   RUNG wire#powerrail
      #MSG[12](MessageType := #CNF, MessageNumber := 12, TraceabilityMode := #Mode, SendMessage := #MSG[14].MessageDone, MasterNFP :=, iNFP := "AutoPositions".St3_Fitting.CodeReadings.SideMemberLH, Data := "AutoPositions".St3_Fitting.CodeReadings.SideMemberRH, Kanban :=, ProcessStatus :=, ErrReset :=, SeqStep :=, oNFP =>, MessageDone => #MessageDone, Answer => #Answer, Fault => #Fault)
   END_RUNG
   // the same network as SCL:
   #MSG[12](MessageType := #CNF,   // "IJCoreMessageProcotol"
            MessageNumber := 12,
            TraceabilityMode := #Mode,
            SendMessage := #MSG[14].MessageDone,
            iNFP := "AutoPositions".St3_Fitting.CodeReadings.SideMemberLH,
            Data := "AutoPositions".St3_Fitting.CodeReadings.SideMemberRH,
            MessageDone => #MessageDone,
            Answer => #Answer,
            Fault => #Fault);
END_REGION

REGION Network 15: MSG013 CNF -13 RearTube
   RUNG wire#powerrail
      #MSG[13](MessageType := #CNF, MessageNumber := 13, TraceabilityMode := #Mode, SendMessage := #MSG[14].MessageDone, MasterNFP :=, iNFP := "AutoPositions".St3_Fitting.CodeReadings.SideMemberLH, Data := "AutoPositions".St3_Fitting.CodeReadings.RearTube, Kanban :=, ProcessStatus :=, ErrReset :=, SeqStep :=, oNFP =>, MessageDone => #MessageDone, Answer => #Answer, Fault => #Fault)
   END_RUNG
   // the same network as SCL:
   #MSG[13](MessageType := #CNF,   // "IJCoreMessageProcotol"
            MessageNumber := 13,
            TraceabilityMode := #Mode,
            SendMessage := #MSG[14].MessageDone,
            iNFP := "AutoPositions".St3_Fitting.CodeReadings.SideMemberLH,
            Data := "AutoPositions".St3_Fitting.CodeReadings.RearTube,
            MessageDone => #MessageDone,
            Answer => #Answer,
            Fault => #Fault);
END_REGION

REGION Network 16: MSG014 PFC 1-1
   RUNG wire#powerrail
      #MSG[14](MessageType := #PFC, MessageNumber := 14, TraceabilityMode := 2, SendMessage :=, MasterNFP :=, iNFP := "AutoPositions".St3_Fitting.CodeReadings.SideMemberLH, Data :=, Kanban := "DB_ProductionProgramActual".Program.FaureciaNumber, ProcessStatus :=, ErrReset :=, SeqStep :=, oNFP =>, MessageDone => #MessageDone, Answer => #Answer, Fault => #Fault)
   END_RUNG
   // the same network as SCL:
   #MSG[14](MessageType := #PFC,   // "IJCoreMessageProcotol"
            MessageNumber := 14,
            TraceabilityMode := 2,
            iNFP := "AutoPositions".St3_Fitting.CodeReadings.SideMemberLH,
            Kanban := "DB_ProductionProgramActual".Program.FaureciaNumber,
            MessageDone => #MessageDone,
            Answer => #Answer,
            Fault => #Fault);
END_REGION

REGION Network 17: MSG015 CNF 1-4 Front Tube
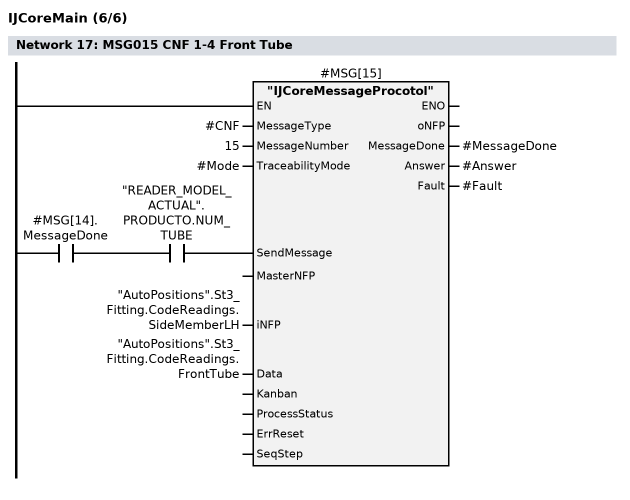
   RUNG wire#powerrail
      #MSG[15](SendMessage := wire#w1, MessageType := #CNF, MessageNumber := 15, TraceabilityMode := #Mode, MasterNFP :=, iNFP := "AutoPositions".St3_Fitting.CodeReadings.SideMemberLH, Data := "AutoPositions".St3_Fitting.CodeReadings.FrontTube, Kanban :=, ProcessStatus :=, ErrReset :=, SeqStep :=, oNFP =>, MessageDone => #MessageDone, Answer => #Answer, Fault => #Fault)
   END_RUNG
   RUNG wire#powerrail
      Contact( #MSG[14].MessageDone )
      Contact( "READER_MODEL_ACTUAL".PRODUCTO.NUM_TUBE )
   END_RUNG wire#w1
   // the same network as SCL:
   #MSG[15](MessageType := #CNF,   // "IJCoreMessageProcotol"
            MessageNumber := 15,
            TraceabilityMode := #Mode,
            SendMessage := #MSG[14].MessageDone AND "READER_MODEL_ACTUAL".PRODUCTO.NUM_TUBE,
            iNFP := "AutoPositions".St3_Fitting.CodeReadings.SideMemberLH,
            Data := "AutoPositions".St3_Fitting.CodeReadings.FrontTube,
            MessageDone => #MessageDone,
            Answer => #Answer,
            Fault => #Fault);
END_REGION
END_FUNCTION_BLOCK

FUNCTION_BLOCK "IJCoreMessageProcotol"
{ S7_Optimized_Access := 'TRUE' }
VERSION : 0.1
   VAR_INPUT 
      MessageType : Int;
      MessageNumber : DInt;
      TraceabilityMode : UInt;
      SendMessage : Bool;
      MasterNFP : Bool;
      iNFP : String;
      Data : String;
      Kanban : String[11];
      ProcessStatus : UInt;
      ErrReset : Bool;
   END_VAR

   VAR_OUTPUT 
      oNFP : String[30];
      MessageDone : Bool;
      Answer : DInt;
      Fault : DInt;
   END_VAR

   VAR_IN_OUT 
      SeqStep : UInt;
   END_VAR

   VAR 
      SEND_OFFSET : Struct
         SW : DInt;
         MSG : DInt;
      END_STRUCT;
      REC_OFFSET : Struct
         SW : DInt;
         MSG : DInt;
         ANS : DInt;
      END_STRUCT;
   END_VAR

   VAR_TEMP 
      i : Int;
   END_VAR

   VAR CONSTANT 
      "DB" : Byte := 16#84;
      CLEAR : Word := 16#0000;
      MINUS1 : Word := 16#FFFF;
      PLUS1 : Word := 16#0001;
      DB_REC : DB_ANY := 1006;
      DB_SEND : DB_ANY := 1005;
      Blank : String := '';
      CNF : Int := 1;
      TRS : Int := 2;
      TRI : Int := 3;
      TRE : Int := 4;
      STA : Int := 5;
      ANDON : Int := 6;
      TRR : Int := 7;
      TRW : Int := 8;
      PFC : Int := 9;
      NFP : Int := 10;
      CMA : Int := 11;
      TMA : Int := 12;
      TRB : Int := 13;
      TRC : Int := 14;
   END_VAR


BEGIN
	//TITLE = 'IJCORE PROTOCOL'
	//AUTHOR: RAUL ROBINS
	//CREATED ON: 03/24/2023
	//VERSION: 3.0
	
	
	
	IF #MessageNumber < 1 OR
	    #MessageType < 0 THEN //If message number 0 end function
	    RETURN;
	END_IF;
	
	
	IF NOT #SendMessage THEN // Error Reset
	    #SeqStep := 0;
	END_IF;
	
	#SEND_OFFSET.SW := (#MessageNumber * 2) + 2; //Calc message send sw offset
	#SEND_OFFSET.MSG := ((#MessageNumber - 1) * 80) + 604; // Calc send message offset
	#REC_OFFSET.SW := (#MessageNumber - 1) * 2; // Calc receive sw offset
	#REC_OFFSET.ANS := ((#MessageNumber - 1) * 32) + 600; // Calc receive answer offset
	#REC_OFFSET.MSG := ((#MessageNumber - 1) * 32) + 602; // Calc receive message offset
	
	
	CASE #SeqStep OF
	    0: // Initial State
	        #MessageDone := FALSE;
	        #Answer := 0;
	        #Fault := 0;
	        POKE(area := #DB, //Clear send flag
	             dbNumber := #DB_SEND,
	             byteOffset := #SEND_OFFSET.SW,
	             value := #MINUS1);
	        POKE(area := #DB, //Clear receive flag
	             dbNumber := #DB_REC,
	             byteOffset := #REC_OFFSET.SW,
	             value := #MINUS1);
	        #oNFP := #Blank;
	        #SeqStep := 10; ///Transition to state 10
	        
	    10: // Wait for start command
	        IF #SendMessage THEN //If start command active
	            
	            #MessageDone := FALSE;
	            #Answer := 0;
	            #Fault := 0;
	            #oNFP := #Blank;
	            
	            POKE(area := #DB, //Clear send flag
	                 dbNumber := #DB_SEND,
	                 byteOffset := #SEND_OFFSET.SW,
	                 value := #MINUS1);
	            POKE(area := #DB, //Clear receive flag
	                 dbNumber := #DB_REC,
	                 byteOffset := #REC_OFFSET.SW,
	                 value := #MINUS1);
	            POKE(area := #DB, // Clear answer 
	                 dbNumber := #DB_REC,
	                 byteOffset := #REC_OFFSET.ANS,
	                 value := #CLEAR);
	            
	            FOR #i := 0 TO 79 BY 1 DO //Clear all send array
	                POKE(area := #DB,
	                     dbNumber := #DB_SEND,
	                     byteOffset := (#SEND_OFFSET.MSG + #i),
	                     value := '$00');
	            END_FOR;
	            FOR #i := 0 TO 29 BY 1 DO //Clear all receive array
	                POKE(area := #DB,
	                     dbNumber := #DB_REC,
	                     byteOffset := (#REC_OFFSET.MSG + #i),
	                     value := '$00');
	            END_FOR;
	            #SeqStep := 20; //Transition to state 20
	        END_IF;
	        
	    20: // Create message to send
	        FOR #i := 0 TO 7 BY 1 DO //Copy NFP to DB to send
	            POKE(area := #DB,
	                 dbNumber := #DB_SEND,
	                 byteOffset := (#SEND_OFFSET.MSG + #i),
	                 value := #iNFP[#i + 1]);
	        END_FOR;
	        CASE #MessageType OF
	                
	                
	            #CNF, #TRB:
	                
	                POKE(area := #DB,
	                     dbNumber := #DB_SEND,
	                     byteOffset := (#SEND_OFFSET.MSG + 8),
	                     value := '7');
	                POKE(area := #DB,
	                     dbNumber := #DB_SEND,
	                     byteOffset := (#SEND_OFFSET.MSG + 9),
	                     value := '0');
	                FOR #i := 0 TO 70 BY 1 DO
	                    POKE(area := #DB,
	                         dbNumber := #DB_SEND,
	                         byteOffset := (#SEND_OFFSET.MSG + #i + 10),
	                         value := #Data[#i + 1]);
	                END_FOR;
	          
	
	                
	            #TRI, #TRR:
	                POKE(area := #DB, //Set the process status of the message
	                     dbNumber := #DB_SEND,
	                     byteOffset := (#SEND_OFFSET.MSG + 8),
	                     value := UINT_TO_CHAR(#ProcessStatus + 48));
	                
	            #STA:
	                FOR #i := 0 TO 7 BY 1 DO //Copy NFP to DB to send
	                    POKE(area := #DB,
	                         dbNumber := #DB_SEND,
	                         byteOffset := (#SEND_OFFSET.MSG + #i),
	                         value := #iNFP[#i + 1]);
	                END_FOR;
	                IF #MasterNFP THEN
	                    #oNFP := #iNFP;
	                END_IF;
	                
	                
	            #PFC:
	                POKE(area := #DB,
	                     dbNumber := #DB_SEND,
	                     byteOffset := (#SEND_OFFSET.MSG + 8),
	                     value := '0');
	                POKE(area := #DB,
	                     dbNumber := #DB_SEND,
	                     byteOffset := (#SEND_OFFSET.MSG + 9),
	                     value := '8');
	                FOR #i := 0 TO 7 BY 1 DO
	                    POKE(area := #DB,
	                         dbNumber := #DB_SEND,
	                         byteOffset := (#SEND_OFFSET.MSG + #i + 10),
	                         value := #Kanban[#i + 1]);
	                END_FOR;
	                
	                
	            #NFP:
	                POKE(area := #DB,
	                     dbNumber := #DB_SEND,
	                     byteOffset := (#SEND_OFFSET.MSG),
	                     value := '0');
	                POKE(area := #DB,
	                     dbNumber := #DB_SEND,
	                     byteOffset := (#SEND_OFFSET.MSG + 1),
	                     value := '8');
	                FOR #i := 1 TO 8 BY 1 DO
	                    POKE(area := #DB,
	                         dbNumber := #DB_SEND,
	                         byteOffset := (#SEND_OFFSET.MSG + #i + 1),
	                         value := #Kanban[#i]);
	                END_FOR;
	                
	            #CMA, #TMA:
	                FOR #i := 0 TO 7 BY 1 DO
	                    POKE(area := #DB,
	                         dbNumber := #DB_SEND,
	                         byteOffset := (#SEND_OFFSET.MSG + #i + 8),
	                         value := #Data[#i + 1]);
	                END_FOR;
	                
	            #TRC:
	                ;
	                
	        END_CASE;
	        
	        
	        
	        #SeqStep := 30; // Transition to state 30
	        
	    30: //Set flag to "1" to inform that PLC is ready to send (DB5 Ó 1005)
	        POKE(area := #DB,//Set flag to "1" to inform that PLC is ready to send
	             dbNumber := #DB_SEND,
	             byteOffset := #SEND_OFFSET.SW,
	             value := #PLUS1);
	        #SeqStep := 40; // Transition to state 40
	        
	        
	    40: //Wait to IJCORE response with "-1"
	        IF (PEEK_WORD(area := #DB, dbNumber := #DB_SEND, byteOffset := #SEND_OFFSET.SW) = #MINUS1)
	        THEN
	            #SeqStep := 50; // Transition to state 50
	        END_IF;
	        
	    50: //Check if IJCORE have answer from DB Receive
	        IF (PEEK_WORD(area := #DB, dbNumber := #DB_REC, byteOffset := #REC_OFFSET.SW) = #PLUS1)
	        THEN
	            #Answer := PEEK_WORD(area := #DB, dbNumber := #DB_REC, byteOffset := #REC_OFFSET.ANS); //Copy answer from IJCORE
	            IF #Answer <> #PLUS1 THEN
	                #Fault := #Answer;
	            END_IF;
	            #SeqStep := 60; // Transition to state 100
	        END_IF;
	        
	    60: //Change Flag to "-1"
	        POKE(area := #DB, //Set "-1" to IJCORE
	             dbNumber := #DB_REC,
	             byteOffset := #REC_OFFSET.SW,
	             value := #MINUS1);
	        #SeqStep := 100; // Transition to state 100
	        
	        
	    100: //Sequence done
	        CASE #TraceabilityMode OF
	            1:// Full traceability
	                IF #Answer = 1 THEN
	                    #MessageDone := TRUE;
	                ELSE
	                    #MessageDone := FALSE;
	                END_IF;
	            2:// Traceability only
	                #MessageDone := TRUE;
	        END_CASE;
	        
	        IF NOT #SendMessage THEN
	            #SeqStep := 0; // Transition to state 0
	        END_IF;
	END_CASE;
	
	
	
	
	
	
	
END_FUNCTION_BLOCK

ORGANIZATION_BLOCK "Startup"   // OB124, LAD, Startup
TITLE = "Complete Restart"
{ S7_Optimized_Access := 'TRUE' }
VERSION : 0.1
// stored: AutoNumber true, IsIECCheckEnabled false, SetENOAutomatically false
   VAR_INPUT
      LostRetentive : Bool;   // True if retentive data are lost
      LostRTC : Bool;   // True if date and time are lost
   END_VAR
BEGIN

REGION Network 1: Braketest or mastering requred
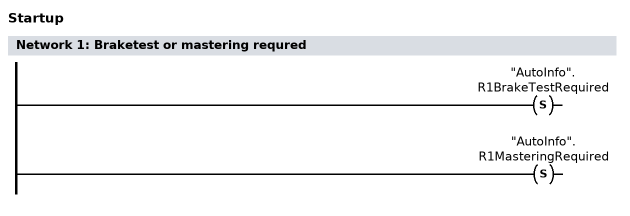
   RUNG wire#powerrail
      S_Coil( "AutoInfo".R1BrakeTestRequired )
   END_RUNG
   RUNG wire#powerrail
      S_Coil( "AutoInfo".R1MasteringRequired )
   END_RUNG
   // the same network as SCL:
   "AutoInfo".R1BrakeTestRequired := TRUE;
   "AutoInfo".R1MasteringRequired := TRUE;
END_REGION

REGION Network 2 (SCL)
       "DevicesData"."TA1-3MA".OverAcc := "StationParameters".Servo.OverAcc;
       "DevicesData"."TA1-3MA".OverDec := "StationParameters".Servo.OverDec;
       "DevicesData"."TA1-3MA".OverV := "StationParameters".Servo.OverV;
       "DevicesData"."TA1-3MA".Velocity := "StationParameters".Servo.Velocity;
END_REGION

REGION Network 3 (SCL)
   "setup_DB".minL := 100.0;
   "setup_DB".minR := "setup_DB".minL;
END_REGION
END_ORGANIZATION_BLOCK

ORGANIZATION_BLOCK "OB_IO_AccessError"   // OB122, LAD, IOAccessError
{ S7_Optimized_Access := 'TRUE' }
VERSION : 0.1
// stored: IsIECCheckEnabled false, SetENOAutomatically false
   VAR_INPUT
      BlockNr : UInt;   // Number of causing block
      Reaction : USInt;   // 0:ignore, 1:substitute, 2:skip
      Fault_ID : Byte;   // 16#42:reading, 16#43:writing
      BlockType : USInt;   // 16#01:OB, 16#02:FC, 16#03:FB, 16#04:SFC, 16#05:SFB, 16#06:DB: Type of block causing the error
      Area : USInt;   // 16#81:I, 16#82:Q: IO area where the IOaccess error occured
      DBNr : DB_ANY;   // Reserved for system
      Csg_OBNr : OB_ANY;   // Number of OB causing the error
      Csg_Prio : USInt;   // Priority of OB causing the error
      Width : USInt;   // 0:bit, 1:byte, 2:word, 3:dword, 4:lword
   END_VAR
BEGIN
END_ORGANIZATION_BLOCK

ORGANIZATION_BLOCK "OB_ProgrammingError"   // OB121, LAD, ProgrammingError
{ S7_Optimized_Access := 'TRUE' }
VERSION : 0.1
// stored: IsIECCheckEnabled false, SetENOAutomatically false
   VAR_INPUT
      BlockNr : UInt;   // Number of causing block
      Reaction : USInt;   // 0:ignore, 1:substitute, 2:skip
      Fault_ID : Byte;   // Fault identifier
      BlockType : USInt;   // 16#01:OB, 16#02:FC, 16#03:FB, 16#04:SFC, 16#05:SFB, 16#06:DB: Type of block causing the error
      Area : USInt;   // Area where the error occured
      DBNr : DB_ANY;   // DB number if Area = DB or DI
      Csg_OBNr : OB_ANY;   // Number of OB causing the error
      Csg_Prio : USInt;   // Priority of OB causing the error
      Width : USInt;   // 0:bit, 1:byte, 2:word, 3:dword, 4:lword
   END_VAR
BEGIN
END_ORGANIZATION_BLOCK

ORGANIZATION_BLOCK "OB_RackStationFailure"   // OB86, LAD, RackOrStationFailure
{ S7_Optimized_Access := 'TRUE' }
VERSION : 0.1
// stored: IsIECCheckEnabled false, SetENOAutomatically false
   VAR_INPUT
      LADDR : HW_DEVICE;   // Hardware identifier
      Event_Class : Byte;   // Event class
      Fault_ID : Byte;   // Fault identifier
   END_VAR
BEGIN
END_ORGANIZATION_BLOCK

ORGANIZATION_BLOCK "OB_Startup"   // OB100, LAD, Startup
TITLE = "Complete Restart"
{ S7_Optimized_Access := 'TRUE' }
VERSION : 0.1
// stored: AutoNumber true, IsIECCheckEnabled false, SetENOAutomatically false
   VAR_INPUT
      LostRetentive : Bool;   // True if retentive data are lost
      LostRTC : Bool;   // True if date and time are lost
   END_VAR
BEGIN
END_ORGANIZATION_BLOCK

FUNCTION_BLOCK "CylinderINC"   // FB30, LAD
{ S7_Optimized_Access := 'FALSE' }
AUTHOR : Bodorik
FAMILY : RIV
NAME : Cylinder
VERSION : 0.9
// stored: AutoNumber false, IsIECCheckEnabled false, SetENOAutomatically false, UDAEnableTagReadback false
   VAR_INPUT
      POWER_OK : Bool;
      MOVE_BASIC : Bool;
      MOVE_WORK : Bool;
      MOVE_FREE : Bool;
      BASIC_POSITION : Bool;
      WORK_POSITION : Bool;
      TRIGGER : Bool;
      RESET : Bool;
      DELAY_BASIC : Time := T#1S;
      DELAY_WORK : Time := T#1S;
      DELAY_FREE : Time := T#1S;
      ERROR_TIME : Time := T#1S;
      ValveDelay : Time;
   END_VAR
   VAR_OUTPUT
      VALVE_BASIC : Bool;
      VALVE_WORK : Bool;
      CylinderStatus : "CylinderStatus";
      ERROR_BASIC : Bool;
      ERROR_WORK : Bool;
   END_VAR
   VAR_IN_OUT
      CylinderOperation : "CylinderOperation";
   END_VAR
   VAR DB_SPECIFIC
      "4l+Started" : Bool;
      InitCommandBP : Bool;
      InitCommandWP : Bool;
      BasicWorkStartWP : Bool;
      BasicWorkStartBP : Bool;
      work_valve : Bool;
      basic_valve : Bool;
      free_valve : Bool;
      baspos_error { S7_SetPoint := 'True'} : TON_TIME;
      workpos_error { S7_SetPoint := 'True'} : TON_TIME;
      baspos_delay { S7_SetPoint := 'True'} : TON_TIME;
      workpos_delay { S7_SetPoint := 'True'} : TON_TIME;
      CylinderOperationOld { S7_SetPoint := 'True'} : "CylinderOperation";
      IEC_Timer_0_Instance { S7_SetPoint := 'True'} : TP_TIME;
   END_VAR
   VAR
      R_TRIG_Instance { S7_SetPoint := 'True'} : R_TRIG;
   END_VAR
   VAR DB_SPECIFIC
      IEC_Timer_0_Instance_1 { S7_SetPoint := 'True'} : TP_TIME;
      IEC_Timer_0_Instance_2 { S7_SetPoint := 'True'} : TP_TIME;
      IEC_Timer_0_Instance_3 { S7_SetPoint := 'True'} : TON_TIME;
      IEC_Timer_0_Instance_4 { S7_SetPoint := 'True'} : TON_TIME;
   END_VAR
   VAR_TEMP
      et : Bool;
   END_VAR
   VAR_TEMP   // added for the SCL form of the ladder/FBD networks
      _w1 : Bool;
   END_VAR
BEGIN

REGION Network 1 (SCL): check new cylinder command
   //check if basic position req movement changed
   IF #CylinderOperation.ToBp <> #CylinderOperationOld.ToBp THEN
       #CylinderOperation.ToFp := false;
       #CylinderOperation.ToWp := false;
   END_IF;
   //check if work position req movement changed
   IF #CylinderOperation.ToWp <> #CylinderOperationOld.ToWp THEN
       #CylinderOperation.ToFp := false;
       #CylinderOperation.ToBp := false;
   END_IF;
   //check if free position req movement changed
   IF #CylinderOperation.ToFp <> #CylinderOperationOld.ToFp THEN
       #CylinderOperation.ToBp := false;
       #CylinderOperation.ToWp := false;
   END_IF;
   //store actual cylinder status to old
   #CylinderOperationOld := #CylinderOperation;
END_REGION

REGION Network 2: Start movement to basic position
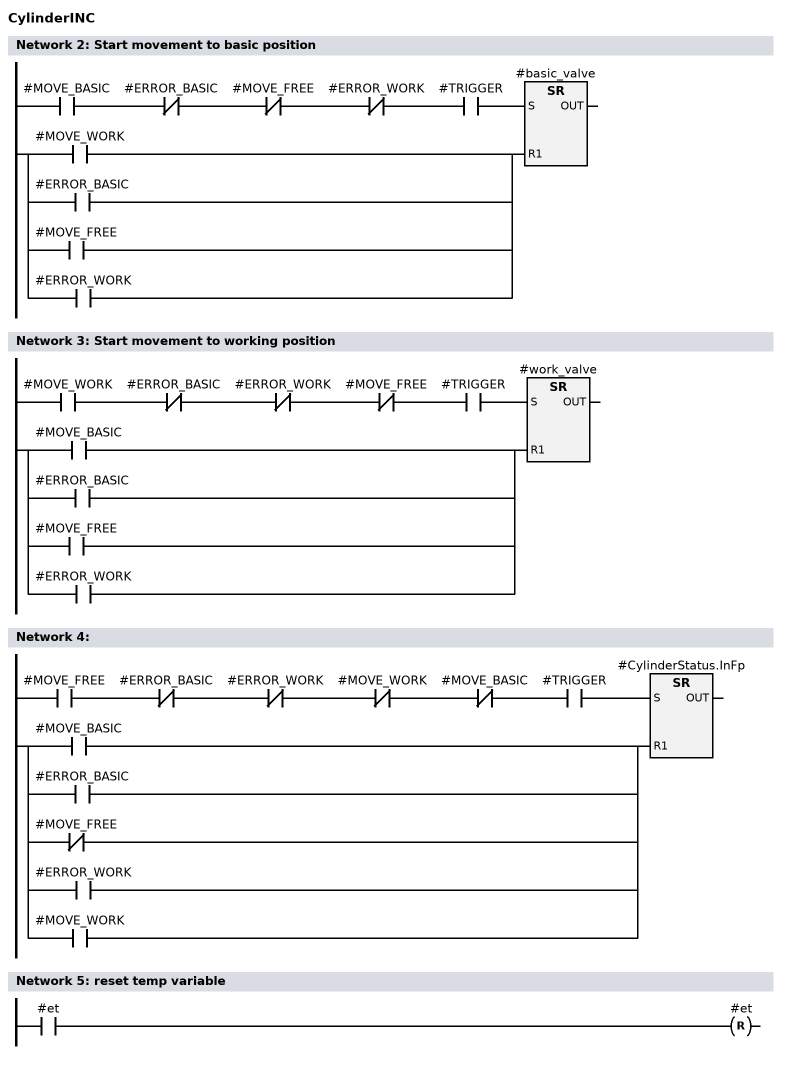
   RUNG wire#powerrail
      Contact( #MOVE_BASIC )
      I_Contact( #ERROR_BASIC )
      I_Contact( #MOVE_FREE )
      I_Contact( #ERROR_WORK )
      Contact( #TRIGGER )
      S_SR(operand := #basic_valve, r1 := wire#w1)
   END_RUNG
   RUNG wire#powerrail
      Contact( #MOVE_WORK )
   END_RUNG wire#w1
   RUNG wire#powerrail
      Contact( #ERROR_BASIC )
   END_RUNG wire#w1
   RUNG wire#powerrail
      Contact( #MOVE_FREE )
   END_RUNG wire#w1
   RUNG wire#powerrail
      Contact( #ERROR_WORK )
   END_RUNG wire#w1
   // the same network as SCL:
   IF #MOVE_BASIC AND NOT #ERROR_BASIC AND NOT #MOVE_FREE AND NOT #ERROR_WORK AND #TRIGGER THEN
       #basic_valve := TRUE;   // SR flip-flop
   END_IF;
   IF #MOVE_WORK OR #ERROR_BASIC OR #MOVE_FREE OR #ERROR_WORK THEN #basic_valve := FALSE; END_IF;
END_REGION

REGION Network 3: Start movement to working position
   RUNG wire#powerrail
      Contact( #MOVE_WORK )
      I_Contact( #ERROR_BASIC )
      I_Contact( #ERROR_WORK )
      I_Contact( #MOVE_FREE )
      Contact( #TRIGGER )
      S_SR(operand := #work_valve, r1 := wire#w1)
   END_RUNG
   RUNG wire#powerrail
      Contact( #MOVE_BASIC )
   END_RUNG wire#w1
   RUNG wire#powerrail
      Contact( #ERROR_BASIC )
   END_RUNG wire#w1
   RUNG wire#powerrail
      Contact( #MOVE_FREE )
   END_RUNG wire#w1
   RUNG wire#powerrail
      Contact( #ERROR_WORK )
   END_RUNG wire#w1
   // the same network as SCL:
   IF #MOVE_WORK AND NOT #ERROR_BASIC AND NOT #ERROR_WORK AND NOT #MOVE_FREE AND #TRIGGER THEN
       #work_valve := TRUE;   // SR flip-flop
   END_IF;
   IF #MOVE_BASIC OR #ERROR_BASIC OR #MOVE_FREE OR #ERROR_WORK THEN #work_valve := FALSE; END_IF;
END_REGION

REGION Network 4
   RUNG wire#powerrail
      Contact( #MOVE_FREE )
      I_Contact( #ERROR_BASIC )
      I_Contact( #ERROR_WORK )
      I_Contact( #MOVE_WORK )
      I_Contact( #MOVE_BASIC )
      Contact( #TRIGGER )
      S_SR(operand := #CylinderStatus.InFp, r1 := wire#w1)
   END_RUNG
   RUNG wire#powerrail
      Contact( #MOVE_BASIC )
   END_RUNG wire#w1
   RUNG wire#powerrail
      Contact( #ERROR_BASIC )
   END_RUNG wire#w1
   RUNG wire#powerrail
      I_Contact( #MOVE_FREE )
   END_RUNG wire#w1
   RUNG wire#powerrail
      Contact( #ERROR_WORK )
   END_RUNG wire#w1
   RUNG wire#powerrail
      Contact( #MOVE_WORK )
   END_RUNG wire#w1
   // the same network as SCL:
   IF #MOVE_FREE AND NOT #ERROR_BASIC AND NOT #ERROR_WORK AND NOT #MOVE_WORK AND NOT #MOVE_BASIC AND #TRIGGER THEN
       #CylinderStatus.InFp := TRUE;   // SR flip-flop
   END_IF;
   IF #MOVE_BASIC OR #ERROR_BASIC OR NOT #MOVE_FREE OR #ERROR_WORK OR #MOVE_WORK THEN
       #CylinderStatus.InFp := FALSE;
   END_IF;
END_REGION

REGION Network 5: reset temp variable
   RUNG wire#powerrail
      Contact( #et )
      R_Coil( #et )
   END_RUNG
   // the same network as SCL:
   IF #et THEN #et := FALSE; END_IF;
END_REGION

REGION Network 6 (FBD): Error movement to basic position
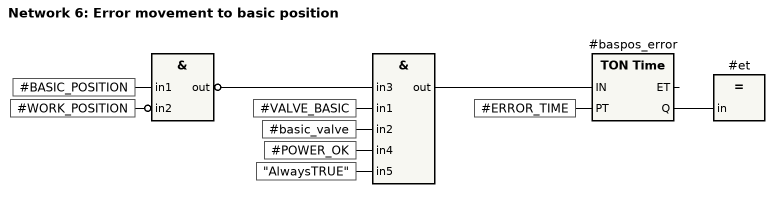
   #baspos_error(IN := NOT (#BASIC_POSITION AND NOT #WORK_POSITION) AND #VALVE_BASIC AND #basic_valve AND #POWER_OK AND "AlwaysTRUE",   // TON
                 PT := #ERROR_TIME);
   #et := #baspos_error.Q;
END_REGION

REGION Network 7: Set basic position error
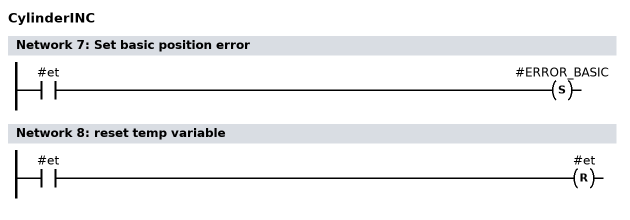
   RUNG wire#powerrail
      Contact( #et )
      S_Coil( #ERROR_BASIC )
   END_RUNG
   // the same network as SCL:
   IF #et THEN #ERROR_BASIC := TRUE; END_IF;
END_REGION

REGION Network 8: reset temp variable
   RUNG wire#powerrail
      Contact( #et )
      R_Coil( #et )
   END_RUNG
   // the same network as SCL:
   IF #et THEN #et := FALSE; END_IF;
END_REGION

REGION Network 9 (FBD): Error movement to working position
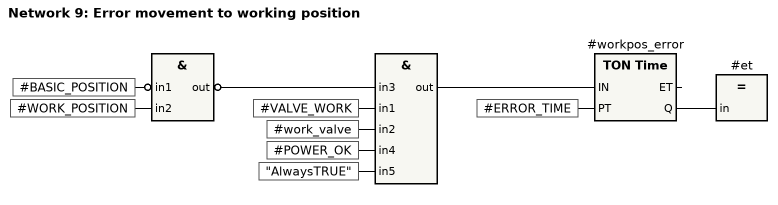
   #workpos_error(IN := NOT (NOT #BASIC_POSITION AND #WORK_POSITION) AND #VALVE_WORK AND #work_valve AND #POWER_OK AND "AlwaysTRUE",   // TON
                  PT := #ERROR_TIME);
   #et := #workpos_error.Q;
END_REGION

REGION Network 10: Set working position error
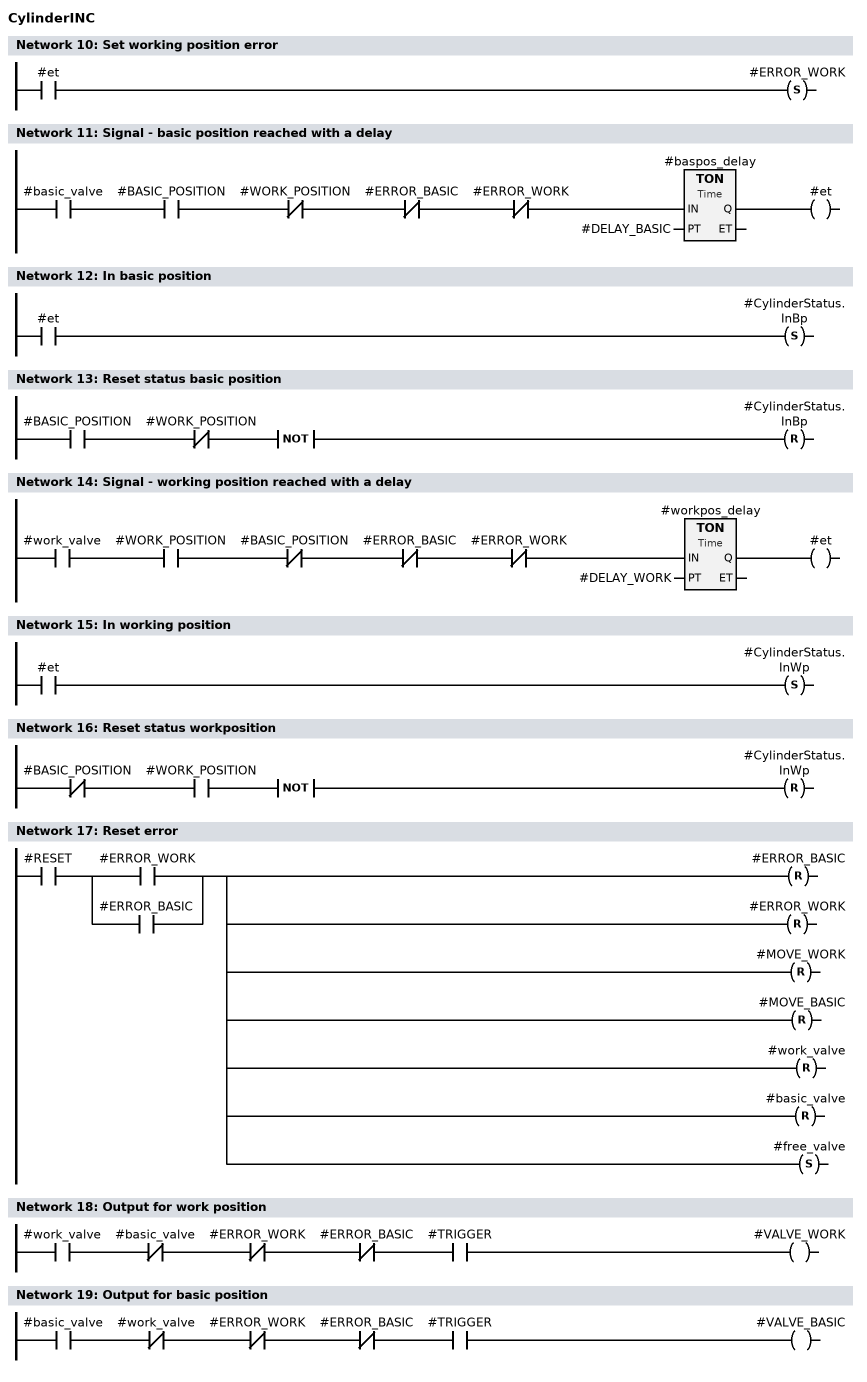
   RUNG wire#powerrail
      Contact( #et )
      S_Coil( #ERROR_WORK )
   END_RUNG
   // the same network as SCL:
   IF #et THEN #ERROR_WORK := TRUE; END_IF;
END_REGION

REGION Network 11: Signal - basic position reached with a delay
   RUNG wire#powerrail
      Contact( #basic_valve )
      Contact( #BASIC_POSITION )
      I_Contact( #WORK_POSITION )
      I_Contact( #ERROR_BASIC )
      I_Contact( #ERROR_WORK )
      { S7_Templates := "time_type := Time" } #baspos_delay.TON(pt := #DELAY_BASIC, et =>)
      Coil( #et )
   END_RUNG
   // the same network as SCL:
   #baspos_delay(PT := #DELAY_BASIC,   // TON
                 IN := #basic_valve AND #BASIC_POSITION AND NOT #WORK_POSITION AND NOT #ERROR_BASIC AND NOT #ERROR_WORK);
   #et := #baspos_delay.Q;
END_REGION

REGION Network 12: In basic position
   RUNG wire#powerrail
      Contact( #et )
      S_Coil( #CylinderStatus.InBp )
   END_RUNG
   // the same network as SCL:
   IF #et THEN #CylinderStatus.InBp := TRUE; END_IF;
END_REGION

REGION Network 13: Reset status basic position
   RUNG wire#powerrail
      Contact( #BASIC_POSITION )
      I_Contact( #WORK_POSITION )
      Not()
      R_Coil( #CylinderStatus.InBp )
   END_RUNG
   // the same network as SCL:
   IF NOT (#BASIC_POSITION AND NOT #WORK_POSITION) THEN #CylinderStatus.InBp := FALSE; END_IF;
END_REGION

REGION Network 14: Signal - working position reached with a delay
   RUNG wire#powerrail
      Contact( #work_valve )
      Contact( #WORK_POSITION )
      I_Contact( #BASIC_POSITION )
      I_Contact( #ERROR_BASIC )
      I_Contact( #ERROR_WORK )
      { S7_Templates := "time_type := Time" } #workpos_delay.TON(pt := #DELAY_WORK, et =>)
      Coil( #et )
   END_RUNG
   // the same network as SCL:
   #workpos_delay(PT := #DELAY_WORK,   // TON
                  IN := #work_valve AND #WORK_POSITION AND NOT #BASIC_POSITION AND NOT #ERROR_BASIC AND NOT #ERROR_WORK);
   #et := #workpos_delay.Q;
END_REGION

REGION Network 15: In working position
   RUNG wire#powerrail
      Contact( #et )
      S_Coil( #CylinderStatus.InWp )
   END_RUNG
   // the same network as SCL:
   IF #et THEN #CylinderStatus.InWp := TRUE; END_IF;
END_REGION

REGION Network 16: Reset status workposition
   RUNG wire#powerrail
      I_Contact( #BASIC_POSITION )
      Contact( #WORK_POSITION )
      Not()
      R_Coil( #CylinderStatus.InWp )
   END_RUNG
   // the same network as SCL:
   IF NOT (NOT #BASIC_POSITION AND #WORK_POSITION) THEN #CylinderStatus.InWp := FALSE; END_IF;
END_REGION

REGION Network 17: Reset error
   RUNG wire#powerrail
      Contact( #RESET )
      wire#w1
      Contact( #ERROR_WORK )
      wire#w2
      R_Coil( #ERROR_BASIC )
   END_RUNG
   RUNG wire#w1
      Contact( #ERROR_BASIC )
   END_RUNG wire#w2
   RUNG wire#w2
      R_Coil( #ERROR_WORK )
   END_RUNG
   RUNG wire#w2
      R_Coil( #MOVE_WORK )
   END_RUNG
   RUNG wire#w2
      R_Coil( #MOVE_BASIC )
   END_RUNG
   RUNG wire#w2
      R_Coil( #work_valve )
   END_RUNG
   RUNG wire#w2
      R_Coil( #basic_valve )
   END_RUNG
   RUNG wire#w2
      S_Coil( #free_valve )
   END_RUNG
   // the same network as SCL:
   #_w1 := #RESET AND (#ERROR_WORK OR #ERROR_BASIC);
   IF #_w1 THEN
       #ERROR_BASIC := FALSE;
       #ERROR_WORK := FALSE;
       #MOVE_WORK := FALSE;
       #MOVE_BASIC := FALSE;
       #work_valve := FALSE;
       #basic_valve := FALSE;
       #free_valve := TRUE;
   END_IF;
END_REGION

REGION Network 18: Output for work position
   RUNG wire#powerrail
      Contact( #work_valve )
      I_Contact( #basic_valve )
      I_Contact( #ERROR_WORK )
      I_Contact( #ERROR_BASIC )
      Contact( #TRIGGER )
      Coil( #VALVE_WORK )
   END_RUNG
   // the same network as SCL:
   #VALVE_WORK := #work_valve AND NOT #basic_valve AND NOT #ERROR_WORK AND NOT #ERROR_BASIC AND #TRIGGER;
END_REGION

REGION Network 19: Output for basic position
   RUNG wire#powerrail
      Contact( #basic_valve )
      I_Contact( #work_valve )
      I_Contact( #ERROR_WORK )
      I_Contact( #ERROR_BASIC )
      Contact( #TRIGGER )
      Coil( #VALVE_BASIC )
   END_RUNG
   // the same network as SCL:
   #VALVE_BASIC := #basic_valve AND NOT #work_valve AND NOT #ERROR_WORK AND NOT #ERROR_BASIC AND #TRIGGER;
END_REGION

REGION Network 20 (SCL)
   #R_TRIG_Instance(CLK:=#POWER_OK
   );

   IF #R_TRIG_Instance.Q THEN
       #"4l+Started" := TRUE;

   END_IF;

   IF #MOVE_BASIC AND #"4l+Started" THEN

       #InitCommandBP := true;
   END_IF;
   IF #MOVE_WORK AND #"4l+Started" THEN

       #InitCommandWP := true;
   END_IF;

   #IEC_Timer_0_Instance_1(IN:=#InitCommandBP,
                               PT:=t#10ms,
                               Q=>#BasicWorkStartBP
       );
   #IEC_Timer_0_Instance_2(IN:=#InitCommandWP,
                               PT:=t#10ms,
                               Q=>#BasicWorkStartWP
   );


   IF #BasicWorkStartBP  THEN
       #VALVE_WORK := TRUE;
       #VALVE_BASIC := FALSE;
       ;

   END_IF;

   IF #BasicWorkStartWP THEN
       #VALVE_WORK := FALSE;
       #VALVE_BASIC := TRUE;
       ;

   END_IF;

   IF NOT #IEC_Timer_0_Instance_1.Q AND #InitCommandBP THEN
       #VALVE_WORK := FALSE;
       #VALVE_BASIC := TRUE;
       #"4l+Started" := FALSE;
       #InitCommandBP := FALSE;
       ;
   END_IF;
   IF NOT #IEC_Timer_0_Instance_2.Q AND #InitCommandWP THEN
       #VALVE_WORK := TRUE;
       #VALVE_BASIC := FALSE;
       #"4l+Started" := FALSE;
       #InitCommandWP := FALSE;
       ;
   END_IF;
END_REGION
END_FUNCTION_BLOCK

FUNCTION "FC_ByteToCharacters" : Void   // FC1071, LAD
{ S7_Optimized_Access := 'FALSE' }
VERSION : 0.1
// stored: AutoNumber false, IsIECCheckEnabled false, SetENOAutomatically false, UDAEnableTagReadback false
   VAR_INPUT
      iByte : Byte;
   END_VAR
   VAR_OUTPUT
      qChar1 : Char;
      qChar2 : Char;
   END_VAR
   VAR_TEMP
      "b" : Byte;
      char1_value : UInt;
      char2_value : UInt;
   END_VAR
   VAR_TEMP   // added for the SCL form of the ladder/FBD networks
      _w1 : Bool;
      _w2 : Bool;
   END_VAR
BEGIN

REGION Network 1: Load input byte to temporary
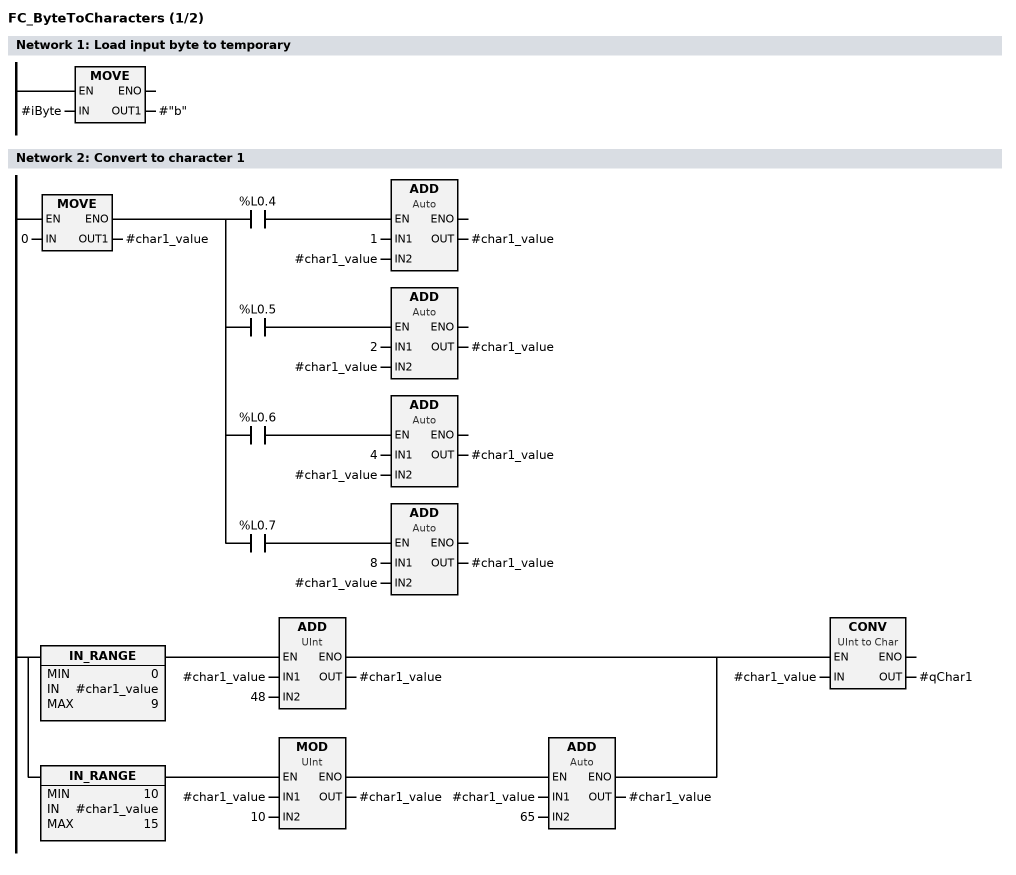
   RUNG wire#powerrail
      Move(in := #iByte, out1 => #"b")
   END_RUNG
   // the same network as SCL:
   #"b" := #iByte;
END_REGION

REGION Network 2: Convert to character 1
   RUNG wire#powerrail
      Move(in := 0, out1 => #char1_value)
      wire#w1
      Contact( %L0.4 )
      Add(in1 := 1, in2 := #char1_value, out => #char1_value)
   END_RUNG
   RUNG wire#w1
      Contact( %L0.5 )
      Add(in1 := 2, in2 := #char1_value, out => #char1_value)
   END_RUNG
   RUNG wire#w1
      Contact( %L0.6 )
      Add(in1 := 4, in2 := #char1_value, out => #char1_value)
   END_RUNG
   RUNG wire#w1
      Contact( %L0.7 )
      Add(in1 := 8, in2 := #char1_value, out => #char1_value)
   END_RUNG
   RUNG wire#powerrail
      { S7_Templates := "SrcType := UInt" } InRange(min := 0, in := #char1_value, max := 9)
      { S7_Templates := "SrcType := UInt" } Add(in1 := #char1_value, in2 := 48, out => #char1_value)
      wire#w2
      { S7_Templates := "[SrcType := UInt, DestType := Char]" } Convert(in := #char1_value, out => #qChar1)
   END_RUNG
   RUNG wire#powerrail
      { S7_Templates := "SrcType := UInt" } InRange(min := 10, in := #char1_value, max := 15)
      { S7_Templates := "SrcType := UInt" } Mod(in1 := #char1_value, in2 := 10, out => #char1_value)
      Add(in1 := #char1_value, in2 := 65, out => #char1_value)
   END_RUNG wire#w2
   // the same network as SCL:
   #char1_value := 0;
   IF %L0.4 THEN #char1_value := 1 + #char1_value; END_IF;
   IF %L0.5 THEN #char1_value := 2 + #char1_value; END_IF;
   IF %L0.6 THEN #char1_value := 4 + #char1_value; END_IF;
   IF %L0.7 THEN #char1_value := 8 + #char1_value; END_IF;
   #_w1 := (0 <= #char1_value) AND (#char1_value <= 9);
   IF #_w1 THEN #char1_value := #char1_value + 48; END_IF;
   #_w2 := (10 <= #char1_value) AND (#char1_value <= 15);
   IF #_w2 THEN
       #char1_value := #char1_value MOD 10;
       #char1_value := #char1_value + 65;
   END_IF;
   IF #_w1 OR #_w2 THEN #qChar1 := UINT_TO_CHAR(#char1_value); END_IF;
END_REGION

REGION Network 3: Convert to character 2
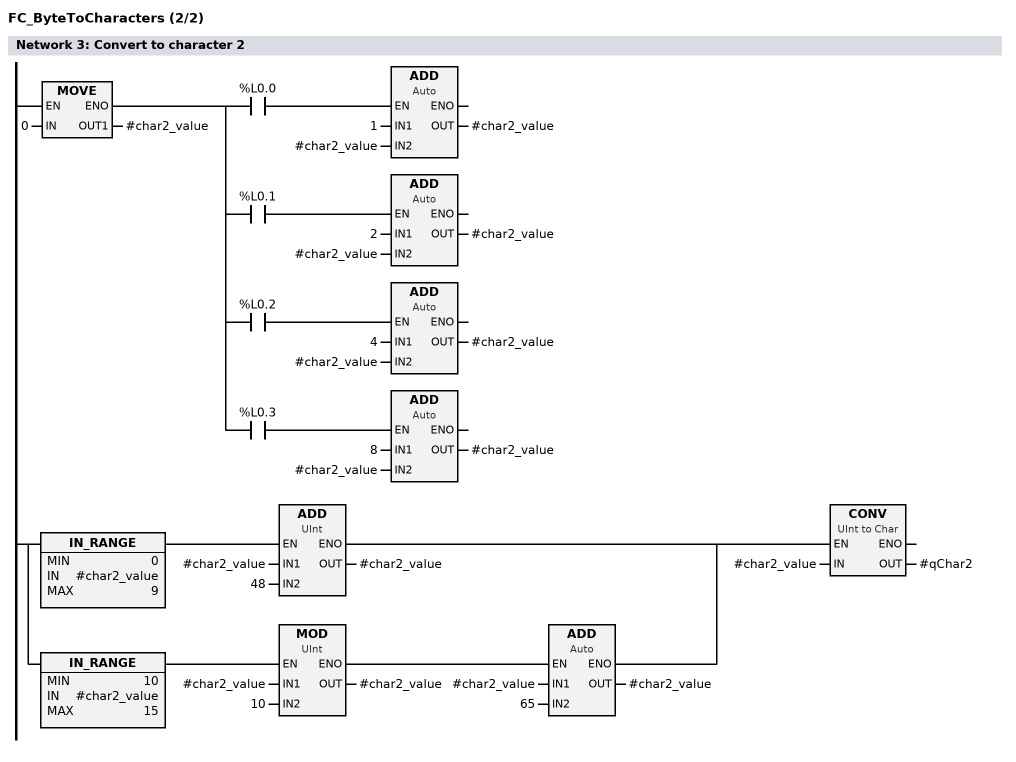
   RUNG wire#powerrail
      Move(in := 0, out1 => #char2_value)
      wire#w1
      Contact( %L0.0 )
      Add(in1 := 1, in2 := #char2_value, out => #char2_value)
   END_RUNG
   RUNG wire#w1
      Contact( %L0.1 )
      Add(in1 := 2, in2 := #char2_value, out => #char2_value)
   END_RUNG
   RUNG wire#w1
      Contact( %L0.2 )
      Add(in1 := 4, in2 := #char2_value, out => #char2_value)
   END_RUNG
   RUNG wire#w1
      Contact( %L0.3 )
      Add(in1 := 8, in2 := #char2_value, out => #char2_value)
   END_RUNG
   RUNG wire#powerrail
      { S7_Templates := "SrcType := UInt" } InRange(min := 0, in := #char2_value, max := 9)
      { S7_Templates := "SrcType := UInt" } Add(in1 := #char2_value, in2 := 48, out => #char2_value)
      wire#w2
      { S7_Templates := "[SrcType := UInt, DestType := Char]" } Convert(in := #char2_value, out => #qChar2)
   END_RUNG
   RUNG wire#powerrail
      { S7_Templates := "SrcType := UInt" } InRange(min := 10, in := #char2_value, max := 15)
      { S7_Templates := "SrcType := UInt" } Mod(in1 := #char2_value, in2 := 10, out => #char2_value)
      Add(in1 := #char2_value, in2 := 65, out => #char2_value)
   END_RUNG wire#w2
   // the same network as SCL:
   #char2_value := 0;
   IF %L0.0 THEN #char2_value := 1 + #char2_value; END_IF;
   IF %L0.1 THEN #char2_value := 2 + #char2_value; END_IF;
   IF %L0.2 THEN #char2_value := 4 + #char2_value; END_IF;
   IF %L0.3 THEN #char2_value := 8 + #char2_value; END_IF;
   #_w1 := (0 <= #char2_value) AND (#char2_value <= 9);
   IF #_w1 THEN #char2_value := #char2_value + 48; END_IF;
   #_w2 := (10 <= #char2_value) AND (#char2_value <= 15);
   IF #_w2 THEN
       #char2_value := #char2_value MOD 10;
       #char2_value := #char2_value + 65;
   END_IF;
   IF #_w1 OR #_w2 THEN #qChar2 := UINT_TO_CHAR(#char2_value); END_IF;
END_REGION
END_FUNCTION

FUNCTION_BLOCK "Main_Safety_RTG1"   // FB0, F_LAD
{ S7_Optimized_Access := 'TRUE' }
VERSION : 0.1
// stored: AutoNumber false, IsIECCheckEnabled false, UDAEnableTagReadback false
   VAR
      ACK_GL_Instance : ACK_GL;
      "ESTOP1_3L+" : ESTOP1;
      "FDBACK_A2.7" : FDBACK;
      "ESTOP1_4L+" : ESTOP1;
      "FDBACK_A2.8" : FDBACK;
      "FDBACK_A2.9" : FDBACK;
      "ESTOP1_5L+" : ESTOP1;
      "F_IEC_Timer_3L+" : TON;
      "F_IEC_Timer_4L+" : TON;
      FDBACK_KF101x : FDBACK;
      FDBACK_KM20_KM21 : FDBACK;
   END_VAR
BEGIN

REGION Network 1: ACK_GL
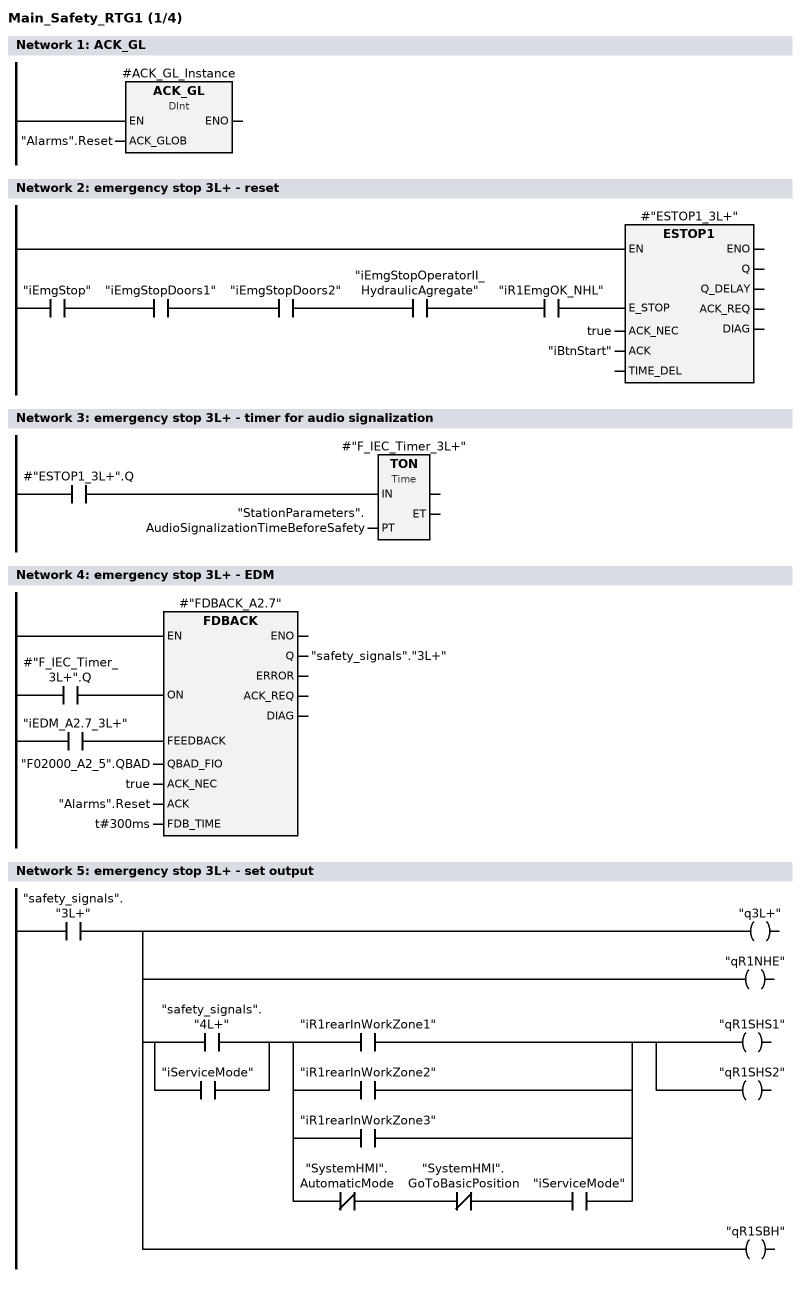
   RUNG wire#powerrail
      { S7_Templates := "codedbool_type := DInt" } #ACK_GL_Instance.ACK_GL(ACK_GLOB := "Alarms".Reset)
   END_RUNG
   // the same network as SCL:
   #ACK_GL_Instance(ACK_GLOB := "Alarms".Reset);   // ACK_GL
END_REGION

REGION Network 2: emergency stop 3L+ - reset
   RUNG wire#powerrail
      #"ESTOP1_3L+".ESTOP1(E_STOP := wire#w1, ACK_NEC := true, ACK := "iBtnStart", TIME_DEL :=, Q =>, Q_DELAY =>, ACK_REQ =>, DIAG =>)
   END_RUNG
   RUNG wire#powerrail
      Contact( "iEmgStop" )
      Contact( "iEmgStopDoors1" )
      Contact( "iEmgStopDoors2" )
      Contact( "iEmgStopOperatorII_HydraulicAgregate" )
      Contact( "iR1EmgOK_NHL" )
   END_RUNG wire#w1
   // the same network as SCL:
   #"ESTOP1_3L+"(E_STOP := "iEmgStop" AND "iEmgStopDoors1" AND "iEmgStopDoors2" AND "iEmgStopOperatorII_HydraulicAgregate" AND "iR1EmgOK_NHL",   // ESTOP1
                 ACK_NEC := true,
                 ACK := "iBtnStart");
END_REGION

REGION Network 3: emergency stop 3L+ - timer for audio signalization
   RUNG wire#powerrail
      Contact( #"ESTOP1_3L+".Q )
      { S7_Templates := "[time_type := Time, codedbool_type := DInt]" } #"F_IEC_Timer_3L+".TON(pt := "StationParameters".AudioSignalizationTimeBeforeSafety, et =>)
   END_RUNG
   // the same network as SCL:
   #"F_IEC_Timer_3L+".TON(IN := #"ESTOP1_3L+".Q, PT := "StationParameters".AudioSignalizationTimeBeforeSafety);
END_REGION

REGION Network 4: emergency stop 3L+ - EDM
   RUNG wire#powerrail
      #"FDBACK_A2.7".FDBACK(ON := wire#w1, FEEDBACK := wire#w2, QBAD_FIO := "F02000_A2_5".QBAD, ACK_NEC := true, ACK := "Alarms".Reset, FDB_TIME := t#300ms, Q => "safety_signals"."3L+", ERROR =>, ACK_REQ =>, DIAG =>)
   END_RUNG
   RUNG wire#powerrail
      Contact( #"F_IEC_Timer_3L+".Q )
   END_RUNG wire#w1
   RUNG wire#powerrail
      Contact( "iEDM_A2.7_3L+" )
   END_RUNG wire#w2
   // the same network as SCL:
   #"FDBACK_A2.7"(ON := #"F_IEC_Timer_3L+".Q,   // FDBACK
                  FEEDBACK := "iEDM_A2.7_3L+",
                  QBAD_FIO := "F02000_A2_5".QBAD,
                  ACK_NEC := true,
                  ACK := "Alarms".Reset,
                  FDB_TIME := t#300ms,
                  Q => "safety_signals"."3L+");
END_REGION

REGION Network 5: emergency stop 3L+ - set output
   RUNG wire#powerrail
      Contact( "safety_signals"."3L+" )
      wire#w1
      Coil( "q3L+" )
   END_RUNG
   RUNG wire#w1
      Coil( "qR1NHE" )
   END_RUNG
   RUNG wire#w1
      Contact( "safety_signals"."4L+" )
      wire#w2
      Contact( "iR1rearInWorkZone1" )
      wire#w3
      Coil( "qR1SHS1" )
   END_RUNG
   RUNG wire#w1
      Contact( "iServiceMode" )
   END_RUNG wire#w2
   RUNG wire#w2
      Contact( "iR1rearInWorkZone2" )
   END_RUNG wire#w3
   RUNG wire#w2
      Contact( "iR1rearInWorkZone3" )
   END_RUNG wire#w3
   RUNG wire#w2
      I_Contact( "SystemHMI".AutomaticMode )
      I_Contact( "SystemHMI".GoToBasicPosition )
      Contact( "iServiceMode" )
   END_RUNG wire#w3
   RUNG wire#w3
      Coil( "qR1SHS2" )
   END_RUNG
   RUNG wire#w1
      Coil( "qR1SBH" )
   END_RUNG
   // the same network as SCL:
   "q3L+" := "safety_signals"."3L+";
   "qR1NHE" := "safety_signals"."3L+";
   "qR1SHS1" := "safety_signals"."3L+" AND ("safety_signals"."4L+" OR "iServiceMode") AND ("iR1rearInWorkZone1" OR "iR1rearInWorkZone2" OR "iR1rearInWorkZone3" OR (NOT "SystemHMI".AutomaticMode AND NOT "SystemHMI".GoToBasicPosition AND "iServiceMode"));
   "qR1SHS2" := "qR1SHS1";
   "qR1SBH" := "safety_signals"."3L+";
END_REGION

REGION Network 6: emergency stop / service doors 4L+ - reset
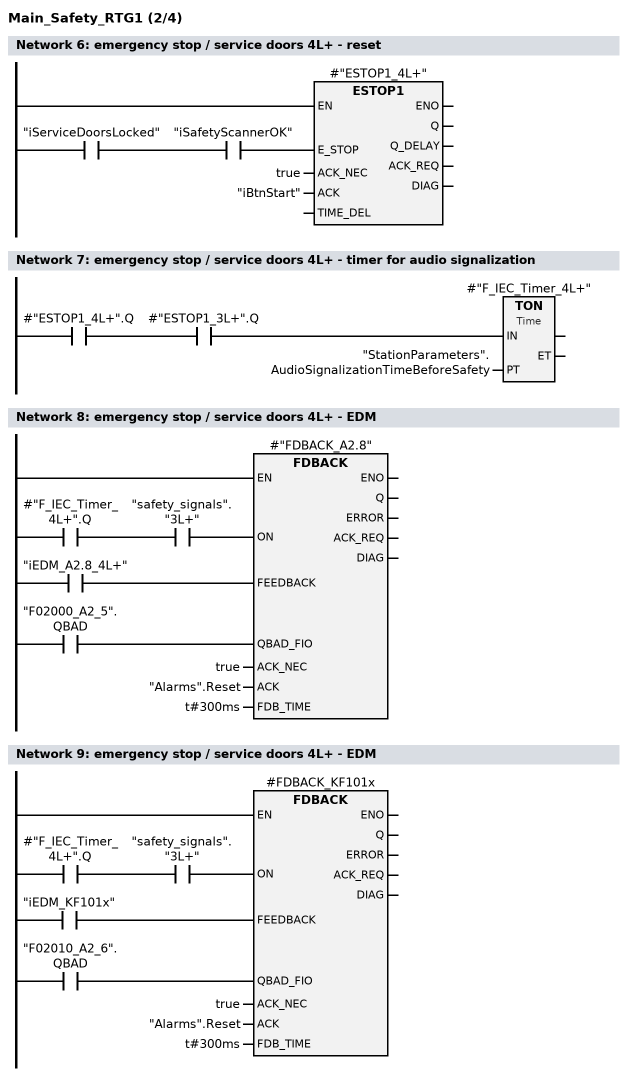
   RUNG wire#powerrail
      #"ESTOP1_4L+".ESTOP1(E_STOP := wire#w1, ACK_NEC := true, ACK := "iBtnStart", TIME_DEL :=, Q =>, Q_DELAY =>, ACK_REQ =>, DIAG =>)
   END_RUNG
   RUNG wire#powerrail
      Contact( "iServiceDoorsLocked" )
      Contact( "iSafetyScannerOK" )
   END_RUNG wire#w1
   // the same network as SCL:
   #"ESTOP1_4L+"(E_STOP := "iServiceDoorsLocked" AND "iSafetyScannerOK", ACK_NEC := true, ACK := "iBtnStart");   // ESTOP1
END_REGION

REGION Network 7: emergency stop / service doors 4L+ - timer for audio signalization
   RUNG wire#powerrail
      Contact( #"ESTOP1_4L+".Q )
      Contact( #"ESTOP1_3L+".Q )
      { S7_Templates := "[time_type := Time, codedbool_type := DInt]" } #"F_IEC_Timer_4L+".TON(pt := "StationParameters".AudioSignalizationTimeBeforeSafety, et =>)
   END_RUNG
   // the same network as SCL:
   #"F_IEC_Timer_4L+".TON(IN := #"ESTOP1_4L+".Q AND #"ESTOP1_3L+".Q,
                          PT := "StationParameters".AudioSignalizationTimeBeforeSafety);
END_REGION

REGION Network 8: emergency stop / service doors 4L+ - EDM
   RUNG wire#powerrail
      #"FDBACK_A2.8".FDBACK(ON := wire#w1, FEEDBACK := wire#w2, QBAD_FIO := wire#w3, ACK_NEC := true, ACK := "Alarms".Reset, FDB_TIME := t#300ms, Q =>, ERROR =>, ACK_REQ =>, DIAG =>)
   END_RUNG
   RUNG wire#powerrail
      Contact( #"F_IEC_Timer_4L+".Q )
      Contact( "safety_signals"."3L+" )
   END_RUNG wire#w1
   RUNG wire#powerrail
      Contact( "iEDM_A2.8_4L+" )
   END_RUNG wire#w2
   RUNG wire#powerrail
      Contact( "F02000_A2_5".QBAD )
   END_RUNG wire#w3
   // the same network as SCL:
   #"FDBACK_A2.8"(ON := #"F_IEC_Timer_4L+".Q AND "safety_signals"."3L+",   // FDBACK
                  FEEDBACK := "iEDM_A2.8_4L+",
                  QBAD_FIO := "F02000_A2_5".QBAD,
                  ACK_NEC := true,
                  ACK := "Alarms".Reset,
                  FDB_TIME := t#300ms);
END_REGION

REGION Network 9: emergency stop / service doors 4L+ - EDM
   RUNG wire#powerrail
      #FDBACK_KF101x.FDBACK(ON := wire#w1, FEEDBACK := wire#w2, QBAD_FIO := wire#w3, ACK_NEC := true, ACK := "Alarms".Reset, FDB_TIME := t#300ms, Q =>, ERROR =>, ACK_REQ =>, DIAG =>)
   END_RUNG
   RUNG wire#powerrail
      Contact( #"F_IEC_Timer_4L+".Q )
      Contact( "safety_signals"."3L+" )
   END_RUNG wire#w1
   RUNG wire#powerrail
      Contact( "iEDM_KF101x" )
   END_RUNG wire#w2
   RUNG wire#powerrail
      Contact( "F02010_A2_6".QBAD )
   END_RUNG wire#w3
   // the same network as SCL:
   #FDBACK_KF101x(ON := #"F_IEC_Timer_4L+".Q AND "safety_signals"."3L+",   // FDBACK
                  FEEDBACK := "iEDM_KF101x",
                  QBAD_FIO := "F02010_A2_6".QBAD,
                  ACK_NEC := true,
                  ACK := "Alarms".Reset,
                  FDB_TIME := t#300ms);
END_REGION

REGION Network 10: emergency stop / service doors 4L+ - set output
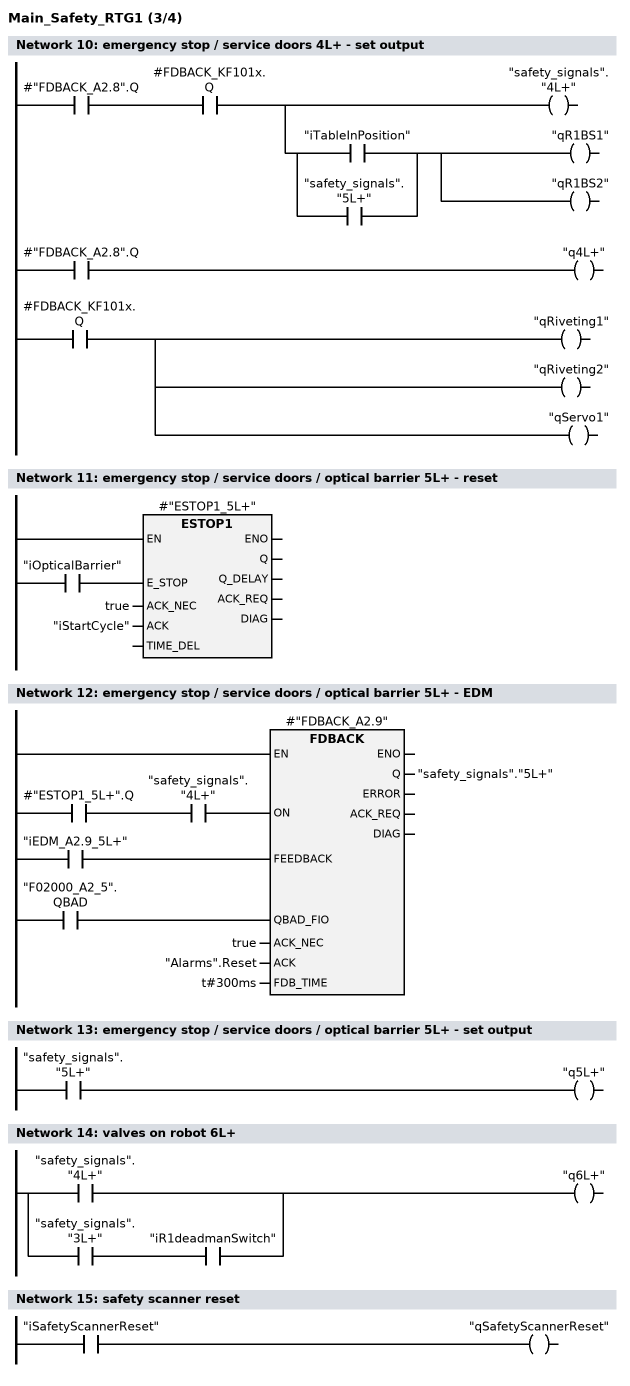
   RUNG wire#powerrail
      Contact( #"FDBACK_A2.8".Q )
      Contact( #FDBACK_KF101x.Q )
      wire#w1
      Coil( "safety_signals"."4L+" )
   END_RUNG
   RUNG wire#w1
      Contact( "iTableInPosition" )
      wire#w2
      Coil( "qR1BS1" )
   END_RUNG
   RUNG wire#w1
      Contact( "safety_signals"."5L+" )
   END_RUNG wire#w2
   RUNG wire#w2
      Coil( "qR1BS2" )
   END_RUNG
   RUNG wire#powerrail
      Contact( #"FDBACK_A2.8".Q )
      Coil( "q4L+" )
   END_RUNG
   RUNG wire#powerrail
      Contact( #FDBACK_KF101x.Q )
      wire#w3
      Coil( "qRiveting1" )
   END_RUNG
   RUNG wire#w3
      Coil( "qRiveting2" )
   END_RUNG
   RUNG wire#w3
      Coil( "qServo1" )
   END_RUNG
   // the same network as SCL:
   "safety_signals"."4L+" := #"FDBACK_A2.8".Q AND #FDBACK_KF101x.Q;
   "qR1BS1" := "safety_signals"."4L+" AND ("iTableInPosition" OR "safety_signals"."5L+");
   "qR1BS2" := "qR1BS1";
   "q4L+" := #"FDBACK_A2.8".Q;
   "qRiveting1" := #FDBACK_KF101x.Q;
   "qRiveting2" := #FDBACK_KF101x.Q;
   "qServo1" := #FDBACK_KF101x.Q;
END_REGION

REGION Network 11: emergency stop / service doors / optical barrier 5L+ - reset
   RUNG wire#powerrail
      #"ESTOP1_5L+".ESTOP1(E_STOP := wire#w1, ACK_NEC := true, ACK := "iStartCycle", TIME_DEL :=, Q =>, Q_DELAY =>, ACK_REQ =>, DIAG =>)
   END_RUNG
   RUNG wire#powerrail
      Contact( "iOpticalBarrier" )
   END_RUNG wire#w1
   // the same network as SCL:
   #"ESTOP1_5L+"(E_STOP := "iOpticalBarrier", ACK_NEC := true, ACK := "iStartCycle");   // ESTOP1
END_REGION

REGION Network 12: emergency stop / service doors / optical barrier 5L+ - EDM
   RUNG wire#powerrail
      #"FDBACK_A2.9".FDBACK(ON := wire#w1, FEEDBACK := wire#w2, QBAD_FIO := wire#w3, ACK_NEC := true, ACK := "Alarms".Reset, FDB_TIME := t#300ms, Q => "safety_signals"."5L+", ERROR =>, ACK_REQ =>, DIAG =>)
   END_RUNG
   RUNG wire#powerrail
      Contact( #"ESTOP1_5L+".Q )
      Contact( "safety_signals"."4L+" )
   END_RUNG wire#w1
   RUNG wire#powerrail
      Contact( "iEDM_A2.9_5L+" )
   END_RUNG wire#w2
   RUNG wire#powerrail
      Contact( "F02000_A2_5".QBAD )
   END_RUNG wire#w3
   // the same network as SCL:
   #"FDBACK_A2.9"(ON := #"ESTOP1_5L+".Q AND "safety_signals"."4L+",   // FDBACK
                  FEEDBACK := "iEDM_A2.9_5L+",
                  QBAD_FIO := "F02000_A2_5".QBAD,
                  ACK_NEC := true,
                  ACK := "Alarms".Reset,
                  FDB_TIME := t#300ms,
                  Q => "safety_signals"."5L+");
END_REGION

REGION Network 13: emergency stop / service doors / optical barrier 5L+ - set output
   RUNG wire#powerrail
      Contact( "safety_signals"."5L+" )
      Coil( "q5L+" )
   END_RUNG
   // the same network as SCL:
   "q5L+" := "safety_signals"."5L+";
END_REGION

REGION Network 14: valves on robot 6L+
   RUNG wire#powerrail
      Contact( "safety_signals"."4L+" )
      wire#w1
      Coil( "q6L+" )
   END_RUNG
   RUNG wire#powerrail
      Contact( "safety_signals"."3L+" )
      Contact( "iR1deadmanSwitch" )
   END_RUNG wire#w1
   // the same network as SCL:
   "q6L+" := "safety_signals"."4L+" OR ("safety_signals"."3L+" AND "iR1deadmanSwitch");
END_REGION

REGION Network 15: safety scanner reset
   RUNG wire#powerrail
      Contact( "iSafetyScannerReset" )
      Coil( "qSafetyScannerReset" )
   END_RUNG
   // the same network as SCL:
   "qSafetyScannerReset" := "iSafetyScannerReset";
END_REGION

REGION Network 16: tool selection for robot - mandatory, but not used
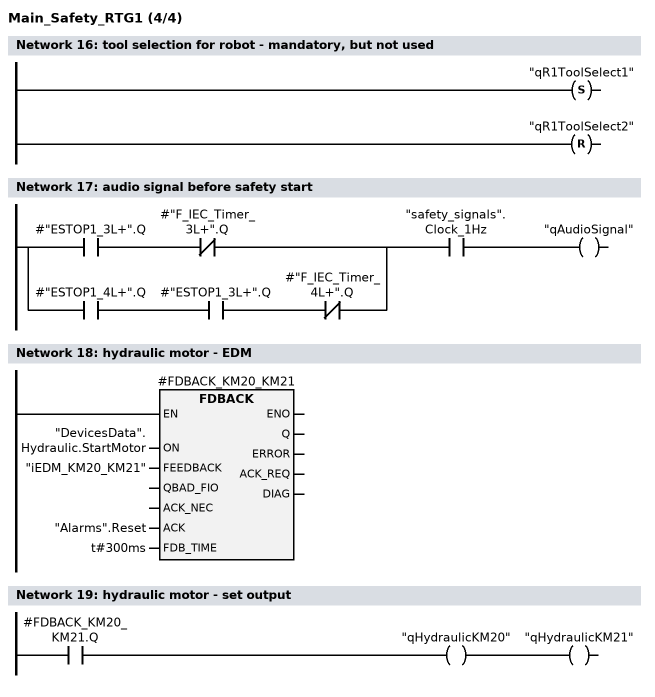
   RUNG wire#powerrail
      S_Coil( "qR1ToolSelect1" )
   END_RUNG
   RUNG wire#powerrail
      R_Coil( "qR1ToolSelect2" )
   END_RUNG
   // the same network as SCL:
   "qR1ToolSelect1" := TRUE;
   "qR1ToolSelect2" := FALSE;
END_REGION

REGION Network 17: audio signal before safety start
   RUNG wire#powerrail
      Contact( #"ESTOP1_3L+".Q )
      I_Contact( #"F_IEC_Timer_3L+".Q )
      wire#w1
      Contact( "safety_signals".Clock_1Hz )
      Coil( "qAudioSignal" )
   END_RUNG
   RUNG wire#powerrail
      Contact( #"ESTOP1_4L+".Q )
      Contact( #"ESTOP1_3L+".Q )
      I_Contact( #"F_IEC_Timer_4L+".Q )
   END_RUNG wire#w1
   // the same network as SCL:
   "qAudioSignal" := ((#"ESTOP1_3L+".Q AND NOT #"F_IEC_Timer_3L+".Q) OR (#"ESTOP1_4L+".Q AND #"ESTOP1_3L+".Q AND NOT #"F_IEC_Timer_4L+".Q)) AND "safety_signals".Clock_1Hz;
END_REGION

REGION Network 18: hydraulic motor - EDM
   RUNG wire#powerrail
      #FDBACK_KM20_KM21.FDBACK(ON := "DevicesData".Hydraulic.StartMotor, FEEDBACK := "iEDM_KM20_KM21", QBAD_FIO :=, ACK_NEC :=, ACK := "Alarms".Reset, FDB_TIME := t#300ms, Q =>, ERROR =>, ACK_REQ =>, DIAG =>)
   END_RUNG
   // the same network as SCL:
   #FDBACK_KM20_KM21(ON := "DevicesData".Hydraulic.StartMotor,   // FDBACK
                     FEEDBACK := "iEDM_KM20_KM21",
                     ACK := "Alarms".Reset,
                     FDB_TIME := t#300ms);
END_REGION

REGION Network 19: hydraulic motor - set output
   RUNG wire#powerrail
      Contact( #FDBACK_KM20_KM21.Q )
      Coil( "qHydraulicKM20" )
      Coil( "qHydraulicKM21" )
   END_RUNG
   // the same network as SCL:
   "qHydraulicKM20" := #FDBACK_KM20_KM21.Q;
   "qHydraulicKM21" := #FDBACK_KM20_KM21.Q;
END_REGION
END_FUNCTION_BLOCK

FUNCTION_BLOCK "sq_autoeject"   // FB53, GRAPH
VERSION : 0.1
// stored: AcknowledgeErrorsRequired true, AutoNumber true, GraphVersion 6.0, InitialValuesAcquisition false, IsIECCheckEnabled false, LanguageInNetworks LAD, LockOperatingMode false, PermanentILProcessingInMANMode false, SetENOAutomatically false, SkipSteps false, UDAEnableTagReadback false, WithAlarmHandling true
   // inherited from GRAPH_BASE
   VAR
      OFF_SQ_BASE : Bool;
   END_VAR
   VAR_INPUT
      OFF_SQ { ExternalWritable := 'False'} : Bool := false;   // Turn sequence off
      INIT_SQ { ExternalWritable := 'False'} : Bool := false;   // Set sequence to initial state
      ACK_EF { ExternalWritable := 'False'} : Bool := false;   // Acknowledge all errors and faults
      S_PREV { ExternalWritable := 'False'} : Bool := false;   // Output previous step in parameter S_NO
      S_NEXT { ExternalWritable := 'False'} : Bool := false;   // Indicate next step in parameter S_NO
      SW_AUTO { ExternalWritable := 'False'} : Bool := false;   // Automatic mode
      SW_TAP { ExternalWritable := 'False'} : Bool := false;   // Semiautomatic/switch with transition
      SW_TOP { ExternalWritable := 'False'} : Bool := false;   // Semiautomatic/ignore transition
      SW_MAN { ExternalWritable := 'False'} : Bool := false;   // Manual mode
      S_SEL { ExternalWritable := 'False'} : Int := 0;   // Select step to be output to S_NO
      S_ON { ExternalWritable := 'False'} : Bool := false;   // Activate step indicated in S_NO
      S_OFF { ExternalWritable := 'False'} : Bool := false;   // Deactivate step indicated S_NO
      T_PUSH { ExternalWritable := 'False'} : Bool := false;   // Enable transition to switch in semi automatic mode
   END_VAR
   VAR_OUTPUT
      S_NO { ExternalWritable := 'False'} : Int := 0;   // Step number
      S_MORE { ExternalWritable := 'False'} : Bool := false;   // More steps are available and can be shown in S_NO
      S_ACTIVE { ExternalWritable := 'False'} : Bool := false;   // Step indicated in S_NO is active
      ERR_FLT { ExternalWritable := 'False'} : Bool := false;   // Interlock or supervision group error
      AUTO_ON { ExternalWritable := 'False'} : Bool := false;   // Automatic mode is active
      TAP_ON { ExternalWritable := 'False'} : Bool := false;   // Semiautomatic mode/step with transition enabled
      TOP_ON { ExternalWritable := 'False'} : Bool := false;   // Semiautomatic mode/ignore transition enabled
      MAN_ON { ExternalWritable := 'False'} : Bool := false;   // Manual mode is active
   END_VAR
   VAR
      dummy : Bool;
      start : Bool;
      base : Bool;
   END_VAR
BEGIN
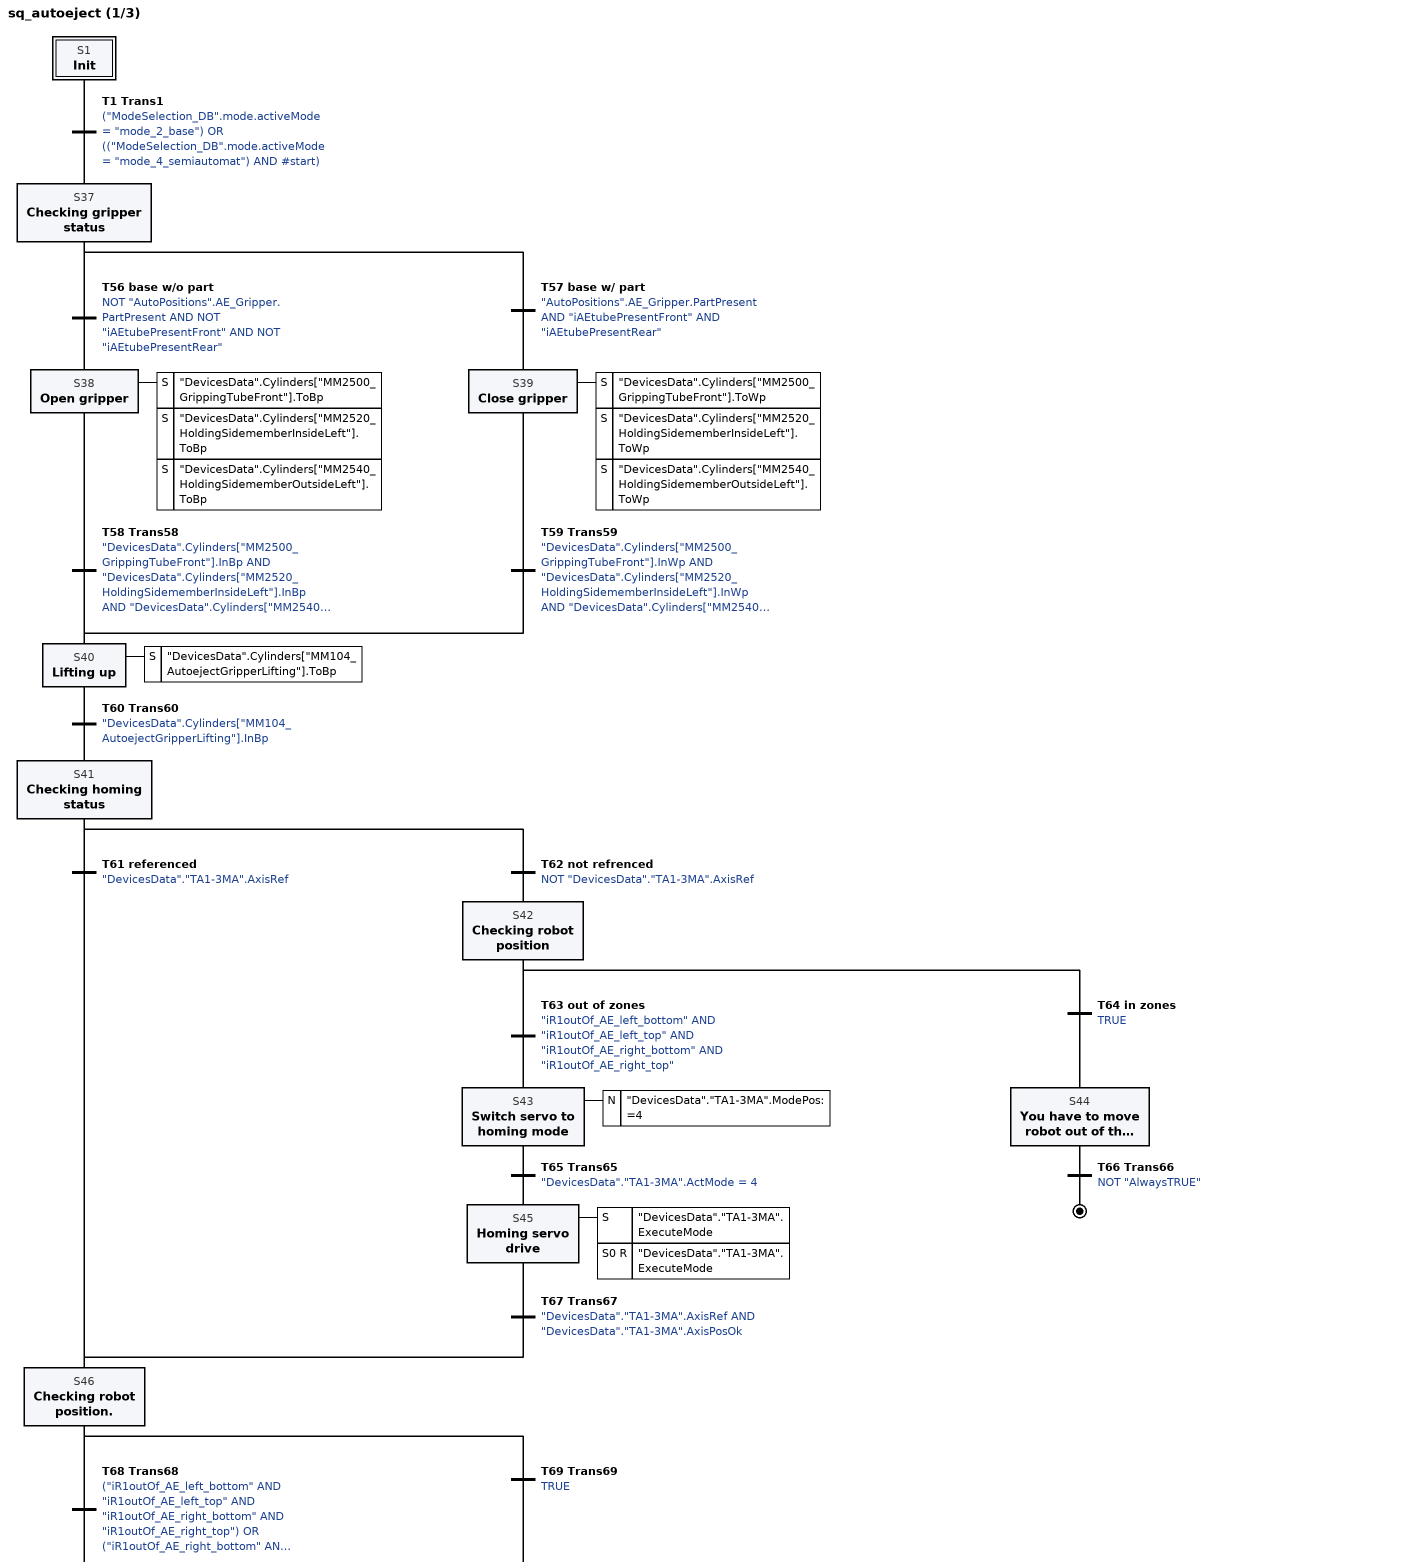
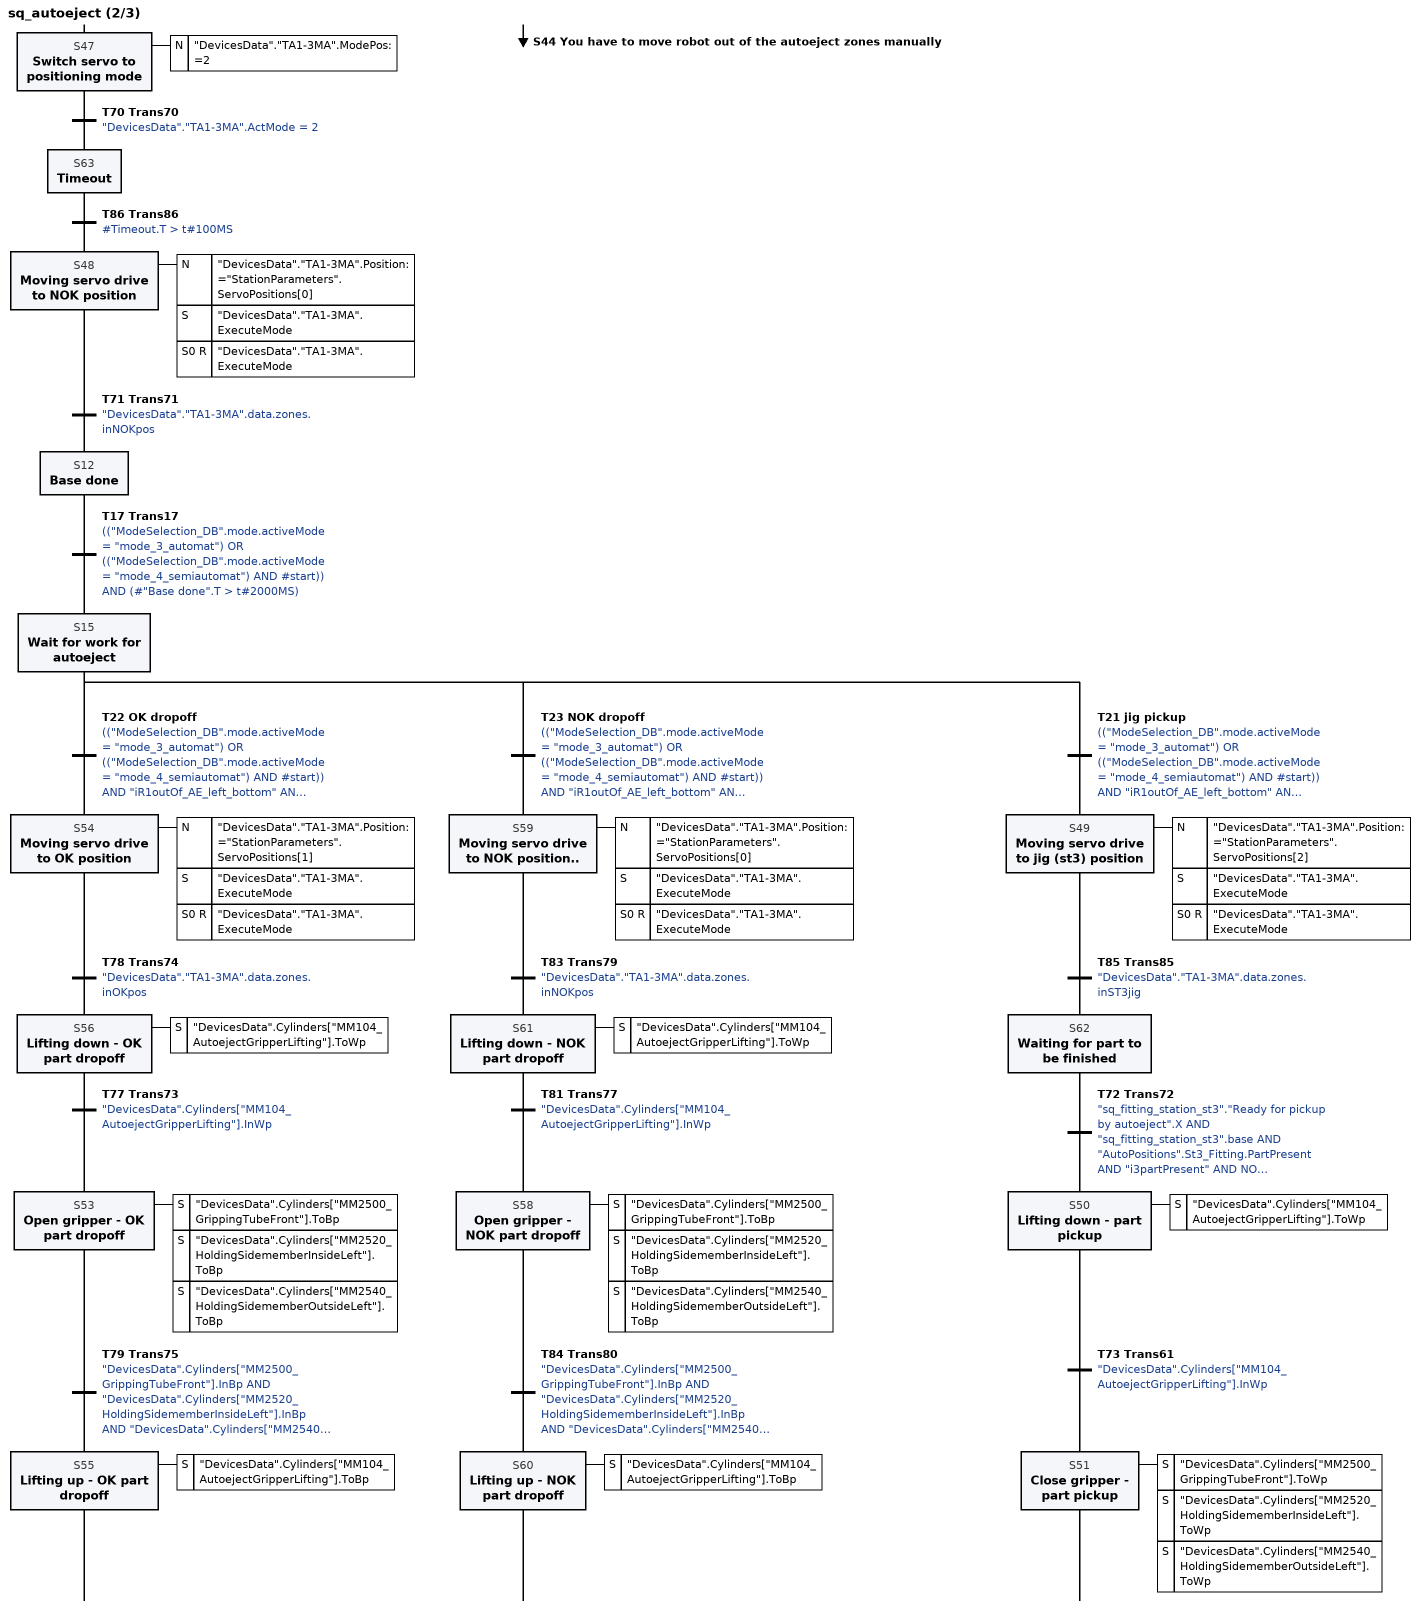
